(* CODESYS project vertical_levitation_control_new.library
   TcLibraryId: TE140x Module Vendor|vertical_levitation_control_new|0.0.0.21
   Company: TE140x Module Vendor
   Title: vertical_levitation_control_new
   Placeholder: vertical_levitation_control_new
   Version: 0.0.0.21

Project tree, tasks and I/O mapping:
  POUs/
    function block FB_vertical_levitation_control_new [ST]: FB_exit, FB_init, nHResult, eInitExceptionHandling, eUpdateExceptionHandling, nExceptionCnt, stActiveException, bInitialized, bExecute
    TcCOM Wrapper/
      function block FB_vertical_levitation_control_new_TcCOM_InitStruct [ST]: FB_init, FB_afterinit, Reinit, FB_exit, eObjectState, nHResult, ipTcComObject, ipADI, nTaskOid, nTaskPriority, nTaskCycleTimeNs, nTaskPort, nTaskSortOrder, eTraceLevelMax, eModuleCaller, eCallerVerification, eStepSizeAdaptation, eExecutionSequence, bExecute, eAccessLockState, eInitExceptionHandling, eUpdateExceptionHandling, stModuleBuildInfo, bInitialized, nSkippedExecutionCount, stLibraryInfo, stModuleInfo, stModuleGeneratorInfo, stSimulinkModelInfo, evertical_levitation_control_new_P_Sharing, nvertical_levitation_control_new_P_Definer, stvertical_levitation_control_new_P, fSimulationTime, nCycleCount, nExceptionCount, stExceptionInfo
  DUTs/
    data type ST_FB_vertical_levitation_control_new_FB_Main
    data type ST_FB_vertical_levitation_control_new_FB_exit
    data type ST_FB_vertical_levitation_control_new_FB_init
    data type ST_GetSet_HRESULT
    data type E_FpExcptCtrlSetEx
    data type ST_GetSet_E_FpExcptCtrlSetEx
    data type ST_GetSet_ULINT
    data type ST_ExceptionInfo
    data type ST_GetSet_ST_ExceptionInfo
    data type ST_GetSet_BOOL
    data type T_matrix3xdouble
    data type T_matrix2xdouble
    data type T_matrix4xdouble
    data type E_SimTimeStep
    data type E_SolverMode
    data type E_ssMatrixType
    data type ST_RTWRTModelMethodsInfo
    data type E_slJmBdControl
    data type ST_ssSolverInfo
    data type T_matrix8xdouble
    data type T_matrix5xdouble
    data type T_matrix4xlogical
    data type T_matrix8xlogical
    data type ST_B_MATLABFunction_vertical_levitation_control_new_T
    data type ST_B_vertical_levitation_control_new_T
    data type T_ZCSigState
    data type T_matrix4xZCSigState
    data type ST_PrevZCX_vertical_levitation_control_new_T
    data type ST_X_vertical_levitation_control_new_T
    data type ST_ExtU_vertical_levitation_control_new_T
    data type ST_ExtY_vertical_levitation_control_new_T
    data type T_matrix4xbool
    data type ST_XDis_vertical_levitation_control_new_T
    data type T_matrix20xdouble
    data type T_matrix20x4xdouble
    data type PLREAL
    data type T_matrix4xdoublepointer
    data type ST_ODE4_IntgData
    data type ST_DW_vertical_levitation_control_new_T
    data type ST_x08a7a7bbd0e5d629f7d70ceec84eacfe
    data type ST_xf09845edab6c83520d8d57def6d6fe1c
    data type ST_RT_MODEL_vertical_levitation_control_new_T
    data type T_matrix53xdouble
    data type T_matrix1007xdouble
    data type T_matrix19xdouble
    data type T_matrix380xdouble
    data type T_matrix3xlogical
    data type ST_P_vertical_levitation_control_new_T
    data type E_ModuleCaller
    data type E_CallerVerification
    data type E_StepSizeAdaptation
    data type E_ExecutionSequence1
    data type E_FpExcptCtrlSet
    data type ST_TcMatSim_ModuleGeneratorInfo
    data type ST_TcMatSim_SimulinkModelInfo
    data type E_ParameterSharingType
    data type ST_FB_vertical_levitation_control_new_TcCOM_InitStruct
    data type ST_FB_vertical_levitation_control_new_TcCOM_InitStruct_FB_init
    data type ST_FB_vertical_levitation_control_new_TcCOM_InitStruct_FB_afterinit
    data type ST_FB_vertical_levitation_control_new_TcCOM_InitStruct_Reinit
    data type ST_FB_vertical_levitation_control_new_TcCOM_InitStruct_FB_Main
    data type ST_FB_vertical_levitation_control_new_TcCOM_InitStruct_FB_exit
    data type ST_GetSet_TCOM_STATE
    data type ST_GetSet_ITComObject
    data type ST_GetSet_ITcADI
    data type ST_vertical_levitation_control_new_U_T
    data type ST_vertical_levitation_control_new_Y_T
    data type ST_vertical_levitation_control_new_X_T
    data type ST_vertical_levitation_control_new_DW_T
    data type ST_GetSet_OTCID
    data type ST_GetSet_UDINT
    data type ST_GetSet_UINT
    data type ST_GetSet_TcTraceLevel
    data type ST_GetSet_E_ModuleCaller
    data type ST_GetSet_E_CallerVerification
    data type ST_GetSet_E_StepSizeAdaptation
    data type ST_GetSet_E_ExecutionSequence1
    data type ST_GetSet_E_FpExcptCtrlSet
    data type ST_ModuleBuildInfo
    data type ST_GetSet_ST_ModuleBuildInfo
    data type ST_LibraryInfo
    data type ST_GetSet_ST_LibraryInfo
    data type ST_ModuleInfo
    data type ST_GetSet_ST_ModuleInfo
    data type ST_GetSet_ST_TcMatSim_ModuleGeneratorInfo
    data type ST_GetSet_ST_TcMatSim_SimulinkModelInfo
    data type ST_GetSet_E_ParameterSharingType
    data type ST_GetSet_ST_P_vertical_levitation_control_new_T
    data type ST_GetSet_LREAL
  Version/
    global variables Global_Version
*)

// DUTs/ST_FB_vertical_levitation_control_new_FB_Main
{attribute 'TcIecLibraryType'}
{attribute 'hide'}
TYPE ST_FB_vertical_levitation_control_new_FB_Main : 
	STRUCT
		{attribute 'GUID' := '18071995-0000-0000-0000-000000000018'}
		pInst : PVOID;
		result : BOOL;
		 {attribute 'hide'}
		_reserved1 : UINT_24_56;
	END_STRUCT
END_TYPE

// DUTs/ST_FB_vertical_levitation_control_new_FB_exit
{attribute 'TcIecLibraryType'}
{attribute 'hide'}
TYPE ST_FB_vertical_levitation_control_new_FB_exit : 
	STRUCT
		{attribute 'GUID' := '18071995-0000-0000-0000-000000000018'}
		pInst : PVOID;
		bInCopyCode : BOOL;
		result : BOOL;
		 {attribute 'hide'}
		_reserved1 : UINT_16_48;
	END_STRUCT
END_TYPE

// DUTs/ST_FB_vertical_levitation_control_new_FB_init
{attribute 'TcIecLibraryType'}
{attribute 'hide'}
TYPE ST_FB_vertical_levitation_control_new_FB_init : 
	STRUCT
		{attribute 'GUID' := '18071995-0000-0000-0000-000000000018'}
		pInst : PVOID;
		bInitRetains : BOOL;
		bInCopyCode : BOOL;
		result : BOOL;
		 {attribute 'hide'}
		_reserved1 : UINT_8_40;
	END_STRUCT
END_TYPE

// DUTs/ST_GetSet_HRESULT
{attribute 'TcIecLibraryType'}
{attribute 'hide'}
TYPE ST_GetSet_HRESULT : 
	STRUCT
		{attribute 'GUID' := '18071995-0000-0000-0000-000000000018'}
		pInst : PVOID;
		{attribute 'GUID' := '18071995-0000-0000-0000-000000000019'}
		nParam : HRESULT;
		 {attribute 'hide'}
		_reserved1 : UINT_0_32;
	END_STRUCT
END_TYPE

// DUTs/E_FpExcptCtrlSetEx
(* Generated from type 'TcMgSdk.FpExcptCtrlSetEx' *)
{attribute 'TcIecLibraryType'}
TYPE E_FpExcptCtrlSetEx : (
	CallerExceptions:=1, 	(* Use the floating point exception settings provided by the caller *)
	ThrowExceptions:=3, 	(* Enable floating point exceptions on invalid operations and divisions by zero *)
	SuppressExceptions:=13, 	(* Disable floating point exceptions. *)
	LogExceptions:=19, 	(* Log exception information. *)
	LogAndHold:=51, 	(* Log exception information and puase execution of the cyclic code after completion of the actual cycle *)
	LogAndCatch:=83, 	(* Log exception information and immediately terminate execution of the cyclic code. Reinitialization is required to restart. *)
	LogAndDump:=147, 	(* Log exception information, create a dump file with detailed exception information and try to continue execution of the cyclic code *)
	LogHoldAndDump:=179, 	(* Log exception information, create a dump file with detailed exception information and puase execution of the cyclic code after completion of the actual cycle *)
	LogCatchAndDump:=211	(* Log exception information, create a dump file with detailed exception information and immediately terminate execution of the cyclic code. Reinitialization is required to restart. *)
) USINT;
END_TYPE

// DUTs/ST_GetSet_E_FpExcptCtrlSetEx
{attribute 'TcIecLibraryType'}
{attribute 'hide'}
TYPE ST_GetSet_E_FpExcptCtrlSetEx : 
	STRUCT
		{attribute 'GUID' := '18071995-0000-0000-0000-000000000018'}
		pInst : PVOID;
		eParam : E_FpExcptCtrlSetEx;
		 {attribute 'hide'}
		_reserved1 : UINT_24_56;
	END_STRUCT
END_TYPE

// DUTs/ST_GetSet_ULINT
{attribute 'TcIecLibraryType'}
{attribute 'hide'}
TYPE ST_GetSet_ULINT : 
	STRUCT
		{attribute 'GUID' := '18071995-0000-0000-0000-000000000018'}
		pInst : PVOID;
		nParam : ULINT;
	END_STRUCT
END_TYPE

// DUTs/ST_ExceptionInfo
(* Generated from type 'TcMgSdk.ExceptionInfo' *)
{attribute 'TcIecLibraryType'}
TYPE ST_ExceptionInfo : 
	STRUCT
		(* Generated from item 'ExceptionCode' *)
		nExceptionCode : DINT;
		(* Generated from item 'TmxName' *)
		{attribute 'GUID' := '18071995-0000-0000-0000-00010000007F'}
		sTmxName : STRING(127);
		(* Generated from item 'TmxVersion' *)
		nTmxVersion : ARRAY [0..3] OF UDINT;
		(* Generated from item 'InstructionAddr' *)
		nInstructionAddr : UDINT;
		(* Generated from item 'ReturnAddr' *)
		nReturnAddr : ARRAY [0..3] OF UDINT;
		(* Generated from item 'DumpCreated' *)
		bDumpCreated : BOOL;
		 {attribute 'hide'}
		_reserved1 : ARRAY [1..3] OF USINT;
	END_STRUCT
END_TYPE

// DUTs/ST_GetSet_ST_ExceptionInfo
{attribute 'TcIecLibraryType'}
{attribute 'hide'}
TYPE ST_GetSet_ST_ExceptionInfo : 
	STRUCT
		{attribute 'GUID' := '18071995-0000-0000-0000-000000000018'}
		pInst : PVOID;
		stParam : ST_ExceptionInfo;
		 {attribute 'hide'}
		_reserved1 : UINT_0_32;
	END_STRUCT
END_TYPE

// DUTs/ST_GetSet_BOOL
{attribute 'TcIecLibraryType'}
{attribute 'hide'}
TYPE ST_GetSet_BOOL : 
	STRUCT
		{attribute 'GUID' := '18071995-0000-0000-0000-000000000018'}
		pInst : PVOID;
		bParam : BOOL;
		 {attribute 'hide'}
		_reserved1 : UINT_24_56;
	END_STRUCT
END_TYPE

// DUTs/T_matrix3xdouble
(* Generated from type 'matrix3xdouble' *)
{attribute 'TcIecLibraryType'}
TYPE T_matrix3xdouble : ARRAY [0..2] OF LREAL;
END_TYPE

// DUTs/T_matrix2xdouble
(* Generated from type 'matrix2xdouble' *)
{attribute 'TcIecLibraryType'}
TYPE T_matrix2xdouble : ARRAY [0..1] OF LREAL;
END_TYPE

// DUTs/T_matrix4xdouble
(* Generated from type 'matrix4xdouble' *)
{attribute 'TcIecLibraryType'}
TYPE T_matrix4xdouble : ARRAY [0..3] OF LREAL;
END_TYPE

// DUTs/E_SimTimeStep
(* Generated from type 'SimTimeStep' *)
{attribute 'TcIecLibraryType'}
{attribute 'qualified_only' := 'true'}
TYPE E_SimTimeStep : (MINOR_TIME_STEP:=0, MAJOR_TIME_STEP:=1) DINT;
END_TYPE

// DUTs/E_SolverMode
(* Generated from type 'SolverMode' *)
{attribute 'TcIecLibraryType'}
{attribute 'qualified_only' := 'true'}
TYPE E_SolverMode : (SOLVER_MODE_AUTO:=0, SOLVER_MODE_SINGLETASKING:=1, SOLVER_MODE_MULTITASKING:=2) DINT;
END_TYPE

// DUTs/E_ssMatrixType
(* Generated from type 'ssMatrixType' *)
{attribute 'TcIecLibraryType'}
{attribute 'qualified_only' := 'true'}
TYPE E_ssMatrixType : (SS_MATRIX_NONE:=0, SS_MATRIX_CONSTANT:=1, SS_MATRIX_TIMEDEP:=2, SS_MATRIX_STATEDEP:=3) DINT;
END_TYPE

// DUTs/ST_RTWRTModelMethodsInfo
(* Generated from type 'RTWRTModelMethodsInfo' *)
{attribute 'TcIecLibraryType'}
TYPE ST_RTWRTModelMethodsInfo : 
	STRUCT
		(* Generated from item 'rtModelPtr' *)
		{attribute 'GUID' := '18071995-0000-0000-0000-000000000018'}
		prtModelPtr : PVOID;
		(* Generated from item 'rtmInitSizesFcn' *)
		{attribute 'GUID' := '18071995-0000-0000-0000-000000000018'}
		prtmInitSizesFcn : PVOID;
		(* Generated from item 'rtmInitSampTimesFcn' *)
		{attribute 'GUID' := '18071995-0000-0000-0000-000000000018'}
		prtmInitSampTimesFcn : PVOID;
		(* Generated from item 'rtmStartFcn' *)
		{attribute 'GUID' := '18071995-0000-0000-0000-000000000018'}
		prtmStartFcn : PVOID;
		(* Generated from item 'rtmOutputsFcn' *)
		{attribute 'GUID' := '18071995-0000-0000-0000-000000000018'}
		prtmOutputsFcn : PVOID;
		(* Generated from item 'rtmUpdateFcn' *)
		{attribute 'GUID' := '18071995-0000-0000-0000-000000000018'}
		prtmUpdateFcn : PVOID;
		(* Generated from item 'rtmDervisFcn' *)
		{attribute 'GUID' := '18071995-0000-0000-0000-000000000018'}
		prtmDervisFcn : PVOID;
		(* Generated from item 'rtmProjectionFcn' *)
		{attribute 'GUID' := '18071995-0000-0000-0000-000000000018'}
		prtmProjectionFcn : PVOID;
		(* Generated from item 'rtmMassMatrixFcn' *)
		{attribute 'GUID' := '18071995-0000-0000-0000-000000000018'}
		prtmMassMatrixFcn : PVOID;
		(* Generated from item 'rtmForcingFunctionFcn' *)
		{attribute 'GUID' := '18071995-0000-0000-0000-000000000018'}
		prtmForcingFunctionFcn : PVOID;
		(* Generated from item 'rtmTerminateFcn' *)
		{attribute 'GUID' := '18071995-0000-0000-0000-000000000018'}
		prtmTerminateFcn : PVOID;
		(* Generated from item 'rtmDiscreteEventsFcn' *)
		{attribute 'GUID' := '18071995-0000-0000-0000-000000000018'}
		prtmDiscreteEventsFcn : PVOID;
	END_STRUCT
END_TYPE

// DUTs/E_slJmBdControl
(* Generated from type 'slJmBdControl' *)
{attribute 'TcIecLibraryType'}
{attribute 'qualified_only' := 'true'}
TYPE E_slJmBdControl : (SL_JM_BD_AUTO:=0, SL_JM_BD_SPARSE_PERTURBATION:=1, SL_JM_BD_FULL_PERTURBATION:=2, SL_JM_BD_SPARSE_ANALYTICAL:=3, SL_JM_BD_FULL_ANALYTICAL:=4) DINT;
END_TYPE

// DUTs/ST_ssSolverInfo
(* Generated from type 'ssSolverInfo' *)
{attribute 'TcIecLibraryType'}
TYPE ST_ssSolverInfo : 
	STRUCT
		(* Generated from item 'rtModelPtr' *)
		{attribute 'GUID' := '18071995-0000-0000-0000-000000000018'}
		prtModelPtr : PVOID;
		simTimeStepPtr : POINTER TO E_SimTimeStep;
		(* Generated from item 'solverData' *)
		{attribute 'GUID' := '18071995-0000-0000-0000-000000000018'}
		psolverData : PVOID;
		solverName : POINTER TO SINT;
		(* Generated from item 'isVariableStepSolver' *)
		bisVariableStepSolver : BOOL;
		(* Generated from item 'solverNeedsReset' *)
		bsolverNeedsReset : BOOL;
		 {attribute 'hide'}
		_reserved1 : UINT;
		(* Generated from item 'solverMode' *)
		esolverMode : E_SolverMode;
		(* Generated from item 'solverStopTime' *)
		fsolverStopTime : LREAL;
		stepSizePtr : POINTER TO LREAL;
		(* Generated from item 'minStepSize' *)
		fminStepSize : LREAL;
		(* Generated from item 'maxStepSize' *)
		fmaxStepSize : LREAL;
		(* Generated from item 'fixedStepSize' *)
		ffixedStepSize : LREAL;
		(* Generated from item 'solverShapePreserveControl' *)
		nsolverShapePreserveControl : DINT;
		(* Generated from item 'solverMaxConsecutiveMinStep' *)
		nsolverMaxConsecutiveMinStep : DINT;
		(* Generated from item 'maxNumMinSteps' *)
		nmaxNumMinSteps : DINT;
		(* Generated from item 'solverMaxOrder' *)
		nsolverMaxOrder : DINT;
		(* Generated from item 'solverConsecutiveZCsStepRelTol' *)
		fsolverConsecutiveZCsStepRelTol : LREAL;
		(* Generated from item 'solverMaxConsecutiveZCs' *)
		nsolverMaxConsecutiveZCs : DINT;
		(* Generated from item 'solverExtrapolationOrder' *)
		nsolverExtrapolationOrder : DINT;
		(* Generated from item 'solverNumberNewtonIterations' *)
		nsolverNumberNewtonIterations : DINT;
		(* Generated from item 'solverRefineFactor' *)
		nsolverRefineFactor : DINT;
		(* Generated from item 'solverRelTol' *)
		fsolverRelTol : LREAL;
		(* Generated from item 'unused_real_T_1' *)
		funused_real_T_1 : LREAL;
		dXPtr : POINTER TO POINTER TO LREAL;
		tPtr : POINTER TO POINTER TO LREAL;
		numContStatesPtr : POINTER TO DINT;
		contStatesPtr : POINTER TO POINTER TO LREAL;
		numPeriodicContStatesPtr : POINTER TO DINT;
		periodicContStateIndicesPtr : POINTER TO POINTER TO DINT;
		periodicContStateRangesPtr : POINTER TO POINTER TO LREAL;
		zcSignalVector : POINTER TO LREAL;
		zcEventsVector : POINTER TO USINT;
		zcSignalAttrib : POINTER TO USINT;
		(* Generated from item 'zcSignalVectorLength' *)
		nzcSignalVectorLength : DINT;
		 {attribute 'hide'}
		_reserved2 : UINT_0_32;
		reserved : POINTER TO USINT;
		(* Generated from item 'foundContZcEvents' *)
		bfoundContZcEvents : BOOL;
		(* Generated from item 'isAtLeftPostOfContZcEvent' *)
		bisAtLeftPostOfContZcEvent : BOOL;
		(* Generated from item 'isAtRightPostOfContZcEvent' *)
		bisAtRightPostOfContZcEvent : BOOL;
		(* Generated from item 'adaptiveZcDetection' *)
		badaptiveZcDetection : BOOL;
		(* Generated from item 'numZcSignals' *)
		nnumZcSignals : DINT;
		(* Generated from item 'stateProjection' *)
		bstateProjection : BOOL;
		(* Generated from item 'robustResetMethod' *)
		brobustResetMethod : BOOL;
		(* Generated from item 'updateJacobianAtReset' *)
		bupdateJacobianAtReset : BOOL;
		(* Generated from item 'consistencyChecking' *)
		bconsistencyChecking : BOOL;
		(* Generated from item 'massMatrixType' *)
		emassMatrixType : E_ssMatrixType;
		(* Generated from item 'massMatrixNzMax' *)
		nmassMatrixNzMax : DINT;
		 {attribute 'hide'}
		_reserved3 : UINT_0_32;
		massMatrixIr : POINTER TO DINT;
		massMatrixJc : POINTER TO DINT;
		massMatrixPr : POINTER TO LREAL;
		errStatusPtr : POINTER TO POINTER TO SINT;
		modelMethodsPtr : POINTER TO ST_RTWRTModelMethodsInfo;
		(* Generated from item 'zcThreshold' *)
		fzcThreshold : LREAL;
		(* Generated from item 'reserved_1' *)
		nreserved_1 : DINT;
		(* Generated from item 'consecutiveZCsError' *)
		nconsecutiveZCsError : DINT;
		(* Generated from item 'CTOutputIncnstWithState' *)
		bCTOutputIncnstWithState : BOOL;
		(* Generated from item 'isComputingJacobian' *)
		bisComputingJacobian : BOOL;
		 {attribute 'hide'}
		_reserved4 : UINT;
		(* Generated from item 'solverJacobianMethodControl' *)
		esolverJacobianMethodControl : E_slJmBdControl;
		(* Generated from item 'ignoredZcDiagnostic' *)
		nignoredZcDiagnostic : DINT;
		(* Generated from item 'maskedZcDiagnostic' *)
		nmaskedZcDiagnostic : DINT;
		(* Generated from item 'isOutputMethodComputed' *)
		bisOutputMethodComputed : BOOL;
		 {attribute 'hide'}
		_reserved5 : ARRAY [1..3] OF USINT;
		(* Generated from item 'maxZcBracketingIterations' *)
		nmaxZcBracketingIterations : DINT;
		(* Generated from item 'isMinorTimeStepWithModeChange' *)
		bisMinorTimeStepWithModeChange : BOOL;
		 {attribute 'hide'}
		_reserved6 : ARRAY [1..3] OF USINT;
		(* Generated from item 'maxZcPerStep' *)
		nmaxZcPerStep : DINT;
		zcSignalPtr : POINTER TO POINTER TO LREAL;
		(* Generated from item 'contStateDisabledPtr' *)
		bcontStateDisabledPtr : POINTER TO POINTER TO BOOL;
		(* Generated from item 'isContModeFrozen' *)
		bisContModeFrozen : BOOL;
		 {attribute 'hide'}
		_reserved7 : ARRAY [1..7] OF USINT;
	END_STRUCT
END_TYPE

// DUTs/T_matrix8xdouble
(* Generated from type 'matrix8xdouble' *)
{attribute 'TcIecLibraryType'}
TYPE T_matrix8xdouble : ARRAY [0..7] OF LREAL;
END_TYPE

// DUTs/T_matrix5xdouble
(* Generated from type 'matrix5xdouble' *)
{attribute 'TcIecLibraryType'}
TYPE T_matrix5xdouble : ARRAY [0..4] OF LREAL;
END_TYPE

// DUTs/T_matrix4xlogical
(* Generated from type 'matrix4xlogical' *)
{attribute 'TcIecLibraryType'}
{attribute 'BaseTypeGUID' := '18071995-0000-0000-0000-000000000030'}
TYPE T_matrix4xlogical : ARRAY [0..3] OF BOOL;
END_TYPE

// DUTs/T_matrix8xlogical
(* Generated from type 'matrix8xlogical' *)
{attribute 'TcIecLibraryType'}
{attribute 'BaseTypeGUID' := '18071995-0000-0000-0000-000000000030'}
TYPE T_matrix8xlogical : ARRAY [0..7] OF BOOL;
END_TYPE

// DUTs/ST_B_MATLABFunction_vertical_levitation_control_new_T
(* Generated from type 'B_MATLABFunction_vertical_levitation_control_new_T' *)
{attribute 'TcIecLibraryType'}
TYPE ST_B_MATLABFunction_vertical_levitation_control_new_T : 
	STRUCT
		(* Generated from item 'y' *)
		ay : T_matrix8xdouble;
	END_STRUCT
END_TYPE

// DUTs/ST_B_vertical_levitation_control_new_T
(* Generated from type 'B_vertical_levitation_control_new_T' *)
{attribute 'TcIecLibraryType'}
TYPE ST_B_vertical_levitation_control_new_T : 
	STRUCT
		(* Generated from item 'UnitDelay' *)
		aUnitDelay : T_matrix4xdouble;
		(* Generated from item 'Switch1' *)
		aSwitch1 : T_matrix4xdouble;
		(* Generated from item 'Switch1_d' *)
		aSwitch1_d : T_matrix4xdouble;
		(* Generated from item 'Gain3' *)
		fGain3 : LREAL;
		(* Generated from item 'Gain7' *)
		fGain7 : LREAL;
		(* Generated from item 'Switch2' *)
		aSwitch2 : T_matrix4xdouble;
		(* Generated from item 'select_maxs' *)
		aselect_maxs : T_matrix4xdouble;
		(* Generated from item 'Delay' *)
		aDelay : T_matrix3xdouble;
		(* Generated from item 'UnitDelay1' *)
		fUnitDelay1 : LREAL;
		(* Generated from item 'FilterCoefficient' *)
		fFilterCoefficient : LREAL;
		(* Generated from item 'Saturation' *)
		fSaturation : LREAL;
		(* Generated from item 'Gain10' *)
		fGain10 : LREAL;
		(* Generated from item 'Integrator' *)
		fIntegrator : LREAL;
		(* Generated from item 'Filtertotgain' *)
		fFiltertotgain : LREAL;
		(* Generated from item 'Add4' *)
		fAdd4 : LREAL;
		(* Generated from item 'UnitDelay1_h' *)
		fUnitDelay1_h : LREAL;
		(* Generated from item 'Add4_f' *)
		fAdd4_f : LREAL;
		(* Generated from item 'UnitDelay1_i' *)
		fUnitDelay1_i : LREAL;
		(* Generated from item 'Add4_d' *)
		fAdd4_d : LREAL;
		(* Generated from item 'UnitDelay1_ie' *)
		fUnitDelay1_ie : LREAL;
		(* Generated from item 'Add4_m' *)
		fAdd4_m : LREAL;
		(* Generated from item 'UnitDelay1_l' *)
		fUnitDelay1_l : LREAL;
		(* Generated from item 'Add4_c' *)
		fAdd4_c : LREAL;
		(* Generated from item 'UnitDelay1_o' *)
		fUnitDelay1_o : LREAL;
		(* Generated from item 'Add4_a' *)
		fAdd4_a : LREAL;
		(* Generated from item 'UnitDelay1_iy' *)
		fUnitDelay1_iy : LREAL;
		(* Generated from item 'Add4_l' *)
		fAdd4_l : LREAL;
		(* Generated from item 'UnitDelay1_a' *)
		fUnitDelay1_a : LREAL;
		(* Generated from item 'Switch1_d5' *)
		fSwitch1_d5 : LREAL;
		(* Generated from item 'Gain12' *)
		fGain12 : LREAL;
		(* Generated from item 'Integrator_g' *)
		fIntegrator_g : LREAL;
		(* Generated from item 'K_D_roll' *)
		fK_D_roll : LREAL;
		(* Generated from item 'Filterrollgain' *)
		fFilterrollgain : LREAL;
		(* Generated from item 'TSamp' *)
		fTSamp : LREAL;
		(* Generated from item 'Diff' *)
		fDiff : LREAL;
		(* Generated from item 'Add4_me' *)
		fAdd4_me : LREAL;
		(* Generated from item 'UnitDelay1_ht' *)
		fUnitDelay1_ht : LREAL;
		(* Generated from item 'Add4_k' *)
		fAdd4_k : LREAL;
		(* Generated from item 'UnitDelay1_oe' *)
		fUnitDelay1_oe : LREAL;
		(* Generated from item 'Add4_ab' *)
		fAdd4_ab : LREAL;
		(* Generated from item 'UnitDelay1_d' *)
		fUnitDelay1_d : LREAL;
		(* Generated from item 'Add4_b' *)
		fAdd4_b : LREAL;
		(* Generated from item 'UnitDelay1_n' *)
		fUnitDelay1_n : LREAL;
		(* Generated from item 'Add4_i' *)
		fAdd4_i : LREAL;
		(* Generated from item 'UnitDelay1_f' *)
		fUnitDelay1_f : LREAL;
		(* Generated from item 'Add4_h' *)
		fAdd4_h : LREAL;
		(* Generated from item 'UnitDelay1_g' *)
		fUnitDelay1_g : LREAL;
		(* Generated from item 'Add4_be' *)
		fAdd4_be : LREAL;
		(* Generated from item 'UnitDelay1_k' *)
		fUnitDelay1_k : LREAL;
		(* Generated from item 'Switch1_m' *)
		fSwitch1_m : LREAL;
		(* Generated from item 'Gain13' *)
		fGain13 : LREAL;
		(* Generated from item 'Integrator_i' *)
		fIntegrator_i : LREAL;
		(* Generated from item 'Filterpitgain' *)
		fFilterpitgain : LREAL;
		(* Generated from item 'Add4_n' *)
		fAdd4_n : LREAL;
		(* Generated from item 'UnitDelay1_fu' *)
		fUnitDelay1_fu : LREAL;
		(* Generated from item 'Add4_g' *)
		fAdd4_g : LREAL;
		(* Generated from item 'UnitDelay1_ha' *)
		fUnitDelay1_ha : LREAL;
		(* Generated from item 'Add4_dq' *)
		fAdd4_dq : LREAL;
		(* Generated from item 'UnitDelay1_ip' *)
		fUnitDelay1_ip : LREAL;
		(* Generated from item 'Add4_dp' *)
		fAdd4_dp : LREAL;
		(* Generated from item 'UnitDelay1_an' *)
		fUnitDelay1_an : LREAL;
		(* Generated from item 'Add4_p' *)
		fAdd4_p : LREAL;
		(* Generated from item 'UnitDelay1_p' *)
		fUnitDelay1_p : LREAL;
		(* Generated from item 'Add4_kw' *)
		fAdd4_kw : LREAL;
		(* Generated from item 'UnitDelay1_dw' *)
		fUnitDelay1_dw : LREAL;
		(* Generated from item 'Add4_hd' *)
		fAdd4_hd : LREAL;
		(* Generated from item 'UnitDelay1_g1' *)
		fUnitDelay1_g1 : LREAL;
		(* Generated from item 'Switch1_n' *)
		fSwitch1_n : LREAL;
		(* Generated from item 'select_mins' *)
		aselect_mins : T_matrix4xdouble;
		(* Generated from item 'Switch' *)
		fSwitch : LREAL;
		(* Generated from item 'UnitDelay1_m' *)
		fUnitDelay1_m : LREAL;
		(* Generated from item 'FilterCoefficient_l' *)
		fFilterCoefficient_l : LREAL;
		(* Generated from item 'Saturation_p' *)
		fSaturation_p : LREAL;
		(* Generated from item 'Switch1_a' *)
		fSwitch1_a : LREAL;
		(* Generated from item 'UnitDelay1_nr' *)
		fUnitDelay1_nr : LREAL;
		(* Generated from item 'FilterCoefficient_o' *)
		fFilterCoefficient_o : LREAL;
		(* Generated from item 'Saturation_pi' *)
		fSaturation_pi : LREAL;
		(* Generated from item 'Switch2_j' *)
		fSwitch2_j : LREAL;
		(* Generated from item 'F_hemsfinal' *)
		aF_hemsfinal : T_matrix4xdouble;
		(* Generated from item 'Switch2_f' *)
		aSwitch2_f : T_matrix8xdouble;
		(* Generated from item 'Switch_o' *)
		fSwitch_o : LREAL;
		(* Generated from item 'Switch_j' *)
		fSwitch_j : LREAL;
		(* Generated from item 'Switch_k' *)
		fSwitch_k : LREAL;
		(* Generated from item 'Add5' *)
		fAdd5 : LREAL;
		(* Generated from item 'Add6' *)
		fAdd6 : LREAL;
		(* Generated from item 'Gain' *)
		fGain : LREAL;
		(* Generated from item 'UnitDelay2' *)
		fUnitDelay2 : LREAL;
		(* Generated from item 'Sum4' *)
		fSum4 : LREAL;
		(* Generated from item 'Sum5' *)
		fSum5 : LREAL;
		(* Generated from item 'Add5_h' *)
		fAdd5_h : LREAL;
		(* Generated from item 'Add6_g' *)
		fAdd6_g : LREAL;
		(* Generated from item 'Gain_l' *)
		fGain_l : LREAL;
		(* Generated from item 'UnitDelay2_k' *)
		fUnitDelay2_k : LREAL;
		(* Generated from item 'Sum4_p' *)
		fSum4_p : LREAL;
		(* Generated from item 'Sum5_p' *)
		fSum5_p : LREAL;
		(* Generated from item 'Add5_m' *)
		fAdd5_m : LREAL;
		(* Generated from item 'Add6_i' *)
		fAdd6_i : LREAL;
		(* Generated from item 'Gain_l5' *)
		fGain_l5 : LREAL;
		(* Generated from item 'UnitDelay2_d' *)
		fUnitDelay2_d : LREAL;
		(* Generated from item 'Sum4_i' *)
		fSum4_i : LREAL;
		(* Generated from item 'Sum5_b' *)
		fSum5_b : LREAL;
		(* Generated from item 'Add5_o' *)
		fAdd5_o : LREAL;
		(* Generated from item 'Add6_m' *)
		fAdd6_m : LREAL;
		(* Generated from item 'Gain_n' *)
		fGain_n : LREAL;
		(* Generated from item 'UnitDelay2_n' *)
		fUnitDelay2_n : LREAL;
		(* Generated from item 'Sum4_f' *)
		fSum4_f : LREAL;
		(* Generated from item 'Sum5_e' *)
		fSum5_e : LREAL;
		(* Generated from item 'Add5_f' *)
		fAdd5_f : LREAL;
		(* Generated from item 'Add6_my' *)
		fAdd6_my : LREAL;
		(* Generated from item 'Gain_ne' *)
		fGain_ne : LREAL;
		(* Generated from item 'UnitDelay2_h' *)
		fUnitDelay2_h : LREAL;
		(* Generated from item 'Sum4_a' *)
		fSum4_a : LREAL;
		(* Generated from item 'Sum5_n' *)
		fSum5_n : LREAL;
		(* Generated from item 'Add5_j' *)
		fAdd5_j : LREAL;
		(* Generated from item 'Add6_l' *)
		fAdd6_l : LREAL;
		(* Generated from item 'Gain_a' *)
		fGain_a : LREAL;
		(* Generated from item 'UnitDelay2_di' *)
		fUnitDelay2_di : LREAL;
		(* Generated from item 'Sum4_pc' *)
		fSum4_pc : LREAL;
		(* Generated from item 'Sum5_g' *)
		fSum5_g : LREAL;
		(* Generated from item 'Add5_k' *)
		fAdd5_k : LREAL;
		(* Generated from item 'Add6_f' *)
		fAdd6_f : LREAL;
		(* Generated from item 'Gain_f' *)
		fGain_f : LREAL;
		(* Generated from item 'UnitDelay2_dw' *)
		fUnitDelay2_dw : LREAL;
		(* Generated from item 'Sum4_d' *)
		fSum4_d : LREAL;
		(* Generated from item 'Sum5_k' *)
		fSum5_k : LREAL;
		(* Generated from item 'Add5_ma' *)
		fAdd5_ma : LREAL;
		(* Generated from item 'Add6_n' *)
		fAdd6_n : LREAL;
		(* Generated from item 'Gain_d' *)
		fGain_d : LREAL;
		(* Generated from item 'UnitDelay2_l' *)
		fUnitDelay2_l : LREAL;
		(* Generated from item 'Sum4_d1' *)
		fSum4_d1 : LREAL;
		(* Generated from item 'Sum5_f' *)
		fSum5_f : LREAL;
		(* Generated from item 'Add5_c' *)
		fAdd5_c : LREAL;
		(* Generated from item 'Add6_mq' *)
		fAdd6_mq : LREAL;
		(* Generated from item 'Gain_k' *)
		fGain_k : LREAL;
		(* Generated from item 'UnitDelay2_o' *)
		fUnitDelay2_o : LREAL;
		(* Generated from item 'Sum4_io' *)
		fSum4_io : LREAL;
		(* Generated from item 'Sum5_j' *)
		fSum5_j : LREAL;
		(* Generated from item 'Add5_op' *)
		fAdd5_op : LREAL;
		(* Generated from item 'Add6_o' *)
		fAdd6_o : LREAL;
		(* Generated from item 'Gain_p' *)
		fGain_p : LREAL;
		(* Generated from item 'UnitDelay2_f' *)
		fUnitDelay2_f : LREAL;
		(* Generated from item 'Sum4_di' *)
		fSum4_di : LREAL;
		(* Generated from item 'Sum5_p3' *)
		fSum5_p3 : LREAL;
		(* Generated from item 'Add5_e' *)
		fAdd5_e : LREAL;
		(* Generated from item 'Add6_k' *)
		fAdd6_k : LREAL;
		(* Generated from item 'Gain_m' *)
		fGain_m : LREAL;
		(* Generated from item 'UnitDelay2_c' *)
		fUnitDelay2_c : LREAL;
		(* Generated from item 'Sum4_e' *)
		fSum4_e : LREAL;
		(* Generated from item 'Sum5_jo' *)
		fSum5_jo : LREAL;
		(* Generated from item 'Add5_kt' *)
		fAdd5_kt : LREAL;
		(* Generated from item 'Add6_d' *)
		fAdd6_d : LREAL;
		(* Generated from item 'Gain_p5' *)
		fGain_p5 : LREAL;
		(* Generated from item 'UnitDelay2_b' *)
		fUnitDelay2_b : LREAL;
		(* Generated from item 'Sum4_c' *)
		fSum4_c : LREAL;
		(* Generated from item 'Sum5_c' *)
		fSum5_c : LREAL;
		(* Generated from item 'Add5_g' *)
		fAdd5_g : LREAL;
		(* Generated from item 'Add6_dl' *)
		fAdd6_dl : LREAL;
		(* Generated from item 'Gain_n2' *)
		fGain_n2 : LREAL;
		(* Generated from item 'UnitDelay2_g' *)
		fUnitDelay2_g : LREAL;
		(* Generated from item 'Sum4_dt' *)
		fSum4_dt : LREAL;
		(* Generated from item 'Sum5_cj' *)
		fSum5_cj : LREAL;
		(* Generated from item 'Add5_gc' *)
		fAdd5_gc : LREAL;
		(* Generated from item 'Add6_a' *)
		fAdd6_a : LREAL;
		(* Generated from item 'Gain_li' *)
		fGain_li : LREAL;
		(* Generated from item 'UnitDelay2_i' *)
		fUnitDelay2_i : LREAL;
		(* Generated from item 'Sum4_k' *)
		fSum4_k : LREAL;
		(* Generated from item 'Sum5_p4' *)
		fSum5_p4 : LREAL;
		(* Generated from item 'Add5_es' *)
		fAdd5_es : LREAL;
		(* Generated from item 'Add6_k2' *)
		fAdd6_k2 : LREAL;
		(* Generated from item 'Gain_i' *)
		fGain_i : LREAL;
		(* Generated from item 'UnitDelay2_n5' *)
		fUnitDelay2_n5 : LREAL;
		(* Generated from item 'Sum4_o' *)
		fSum4_o : LREAL;
		(* Generated from item 'Sum5_po' *)
		fSum5_po : LREAL;
		(* Generated from item 'Add5_l' *)
		fAdd5_l : LREAL;
		(* Generated from item 'Add6_c' *)
		fAdd6_c : LREAL;
		(* Generated from item 'Gain_mr' *)
		fGain_mr : LREAL;
		(* Generated from item 'UnitDelay2_e' *)
		fUnitDelay2_e : LREAL;
		(* Generated from item 'Sum4_p3' *)
		fSum4_p3 : LREAL;
		(* Generated from item 'Sum5_nz' *)
		fSum5_nz : LREAL;
		(* Generated from item 'Add5_je' *)
		fAdd5_je : LREAL;
		(* Generated from item 'Add6_a2' *)
		fAdd6_a2 : LREAL;
		(* Generated from item 'Gain_fh' *)
		fGain_fh : LREAL;
		(* Generated from item 'UnitDelay2_cg' *)
		fUnitDelay2_cg : LREAL;
		(* Generated from item 'Sum4_o5' *)
		fSum4_o5 : LREAL;
		(* Generated from item 'Sum5_d' *)
		fSum5_d : LREAL;
		(* Generated from item 'Add5_b' *)
		fAdd5_b : LREAL;
		(* Generated from item 'Add6_e' *)
		fAdd6_e : LREAL;
		(* Generated from item 'Gain_j' *)
		fGain_j : LREAL;
		(* Generated from item 'UnitDelay2_c5' *)
		fUnitDelay2_c5 : LREAL;
		(* Generated from item 'Sum4_fb' *)
		fSum4_fb : LREAL;
		(* Generated from item 'Sum5_js' *)
		fSum5_js : LREAL;
		(* Generated from item 'Add5_b0' *)
		fAdd5_b0 : LREAL;
		(* Generated from item 'Add6_nn' *)
		fAdd6_nn : LREAL;
		(* Generated from item 'Gain_pn' *)
		fGain_pn : LREAL;
		(* Generated from item 'UnitDelay2_k0' *)
		fUnitDelay2_k0 : LREAL;
		(* Generated from item 'Sum4_pd' *)
		fSum4_pd : LREAL;
		(* Generated from item 'Sum5_m' *)
		fSum5_m : LREAL;
		(* Generated from item 'Add5_fq' *)
		fAdd5_fq : LREAL;
		(* Generated from item 'Add6_i1' *)
		fAdd6_i1 : LREAL;
		(* Generated from item 'Gain_p0' *)
		fGain_p0 : LREAL;
		(* Generated from item 'UnitDelay2_o4' *)
		fUnitDelay2_o4 : LREAL;
		(* Generated from item 'Sum4_kn' *)
		fSum4_kn : LREAL;
		(* Generated from item 'Sum5_a' *)
		fSum5_a : LREAL;
		(* Generated from item 'Add5_mq' *)
		fAdd5_mq : LREAL;
		(* Generated from item 'Add6_j' *)
		fAdd6_j : LREAL;
		(* Generated from item 'Gain_ay' *)
		fGain_ay : LREAL;
		(* Generated from item 'UnitDelay2_hz' *)
		fUnitDelay2_hz : LREAL;
		(* Generated from item 'Sum4_ku' *)
		fSum4_ku : LREAL;
		(* Generated from item 'Sum5_kh' *)
		fSum5_kh : LREAL;
		(* Generated from item 'IsPeak1' *)
		aIsPeak1 : T_matrix4xdouble;
		(* Generated from item 'Switch2_d' *)
		aSwitch2_d : T_matrix4xdouble;
		(* Generated from item 'F_netpostfm' *)
		aF_netpostfm : T_matrix3xdouble;
		(* Generated from item 'Sum' *)
		fSum : LREAL;
		(* Generated from item 'Sum1' *)
		fSum1 : LREAL;
		(* Generated from item 'clamppit' *)
		fclamppit : LREAL;
		(* Generated from item 'Sum_f' *)
		fSum_f : LREAL;
		(* Generated from item 'Sum1_a' *)
		fSum1_a : LREAL;
		(* Generated from item 'clamproll' *)
		fclamproll : LREAL;
		(* Generated from item 'clamptot' *)
		fclamptot : LREAL;
		(* Generated from item 'K_I_tot' *)
		fK_I_tot : LREAL;
		(* Generated from item 'K_I_roll' *)
		fK_I_roll : LREAL;
		(* Generated from item 'K_I_pit' *)
		fK_I_pit : LREAL;
		(* Generated from item 'current_reqf' *)
		fcurrent_reqf : LREAL;
		(* Generated from item 'current_reqb' *)
		fcurrent_reqb : LREAL;
		(* Generated from item 'current_reqf_p' *)
		fcurrent_reqf_p : LREAL;
		(* Generated from item 'current_reqb_o' *)
		fcurrent_reqb_o : LREAL;
		(* Generated from item 'current_reqf_c' *)
		fcurrent_reqf_c : LREAL;
		(* Generated from item 'current_reqb_c' *)
		fcurrent_reqb_c : LREAL;
		(* Generated from item 'current_reqf_h' *)
		fcurrent_reqf_h : LREAL;
		(* Generated from item 'current_reqb_e' *)
		fcurrent_reqb_e : LREAL;
		(* Generated from item 'F_hems' *)
		aF_hems : T_matrix4xdouble;
		(* Generated from item 'Switch2_l' *)
		aSwitch2_l : T_matrix4xdouble;
		(* Generated from item 'Sum5_fo' *)
		fSum5_fo : LREAL;
		(* Generated from item 'Is' *)
		aIs : T_matrix4xdouble;
		(* Generated from item 'satn' *)
		asatn : T_matrix8xdouble;
		(* Generated from item 'airgaps_avg' *)
		aairgaps_avg : T_matrix4xdouble;
		(* Generated from item 'airgap_diff' *)
		fairgap_diff : LREAL;
		(* Generated from item 'tau_x' *)
		ftau_x : LREAL;
		(* Generated from item 'corrected_out' *)
		fcorrected_out : LREAL;
		(* Generated from item 'corrected_out_j' *)
		fcorrected_out_j : LREAL;
		(* Generated from item 'corrected_out_o' *)
		fcorrected_out_o : LREAL;
		(* Generated from item 'F_hems_b' *)
		aF_hems_b : T_matrix4xdouble;
		(* Generated from item 'clamp_tot' *)
		aclamp_tot : T_matrix2xdouble;
		(* Generated from item 'clamp_roll' *)
		aclamp_roll : T_matrix2xdouble;
		(* Generated from item 'clamp_pit' *)
		aclamp_pit : T_matrix2xdouble;
		(* Generated from item 'counter' *)
		acounter : T_matrix5xdouble;
		(* Generated from item 'F_dof_sat' *)
		aF_dof_sat : T_matrix3xdouble;
		(* Generated from item 'sat_fail' *)
		fsat_fail : LREAL;
		(* Generated from item 'q' *)
		fq : LREAL;
		(* Generated from item 'q_c' *)
		fq_c : LREAL;
		(* Generated from item 'q_k' *)
		fq_k : LREAL;
		(* Generated from item 'q_i' *)
		fq_i : LREAL;
		(* Generated from item 'q_g' *)
		fq_g : LREAL;
		(* Generated from item 'q_ke' *)
		fq_ke : LREAL;
		(* Generated from item 'q_b' *)
		fq_b : LREAL;
		(* Generated from item 'q_km' *)
		fq_km : LREAL;
		(* Generated from item 'q_o' *)
		fq_o : LREAL;
		(* Generated from item 'q_a' *)
		fq_a : LREAL;
		(* Generated from item 'q_ag' *)
		fq_ag : LREAL;
		(* Generated from item 'q_d' *)
		fq_d : LREAL;
		(* Generated from item 'q_f' *)
		fq_f : LREAL;
		(* Generated from item 'q_m' *)
		fq_m : LREAL;
		(* Generated from item 'q_n' *)
		fq_n : LREAL;
		(* Generated from item 'q_iy' *)
		fq_iy : LREAL;
		(* Generated from item 'q_h' *)
		fq_h : LREAL;
		(* Generated from item 'q_kmf' *)
		fq_kmf : LREAL;
		(* Generated from item 'q_a3' *)
		fq_a3 : LREAL;
		(* Generated from item 'q_ac' *)
		fq_ac : LREAL;
		(* Generated from item 'q_p' *)
		fq_p : LREAL;
		(* Generated from item 'UnaryMinus' *)
		fUnaryMinus : LREAL;
		(* Generated from item 'UnaryMinus_l' *)
		fUnaryMinus_l : LREAL;
		(* Generated from item 'UnaryMinus_k' *)
		fUnaryMinus_k : LREAL;
		(* Generated from item 'UnaryMinus_b' *)
		fUnaryMinus_b : LREAL;
		(* Generated from item 'UnaryMinus_d' *)
		fUnaryMinus_d : LREAL;
		(* Generated from item 'UnaryMinus_f' *)
		fUnaryMinus_f : LREAL;
		(* Generated from item 'UnaryMinus_k2' *)
		fUnaryMinus_k2 : LREAL;
		(* Generated from item 'UnaryMinus_dc' *)
		fUnaryMinus_dc : LREAL;
		(* Generated from item 'UnaryMinus_m' *)
		fUnaryMinus_m : LREAL;
		(* Generated from item 'UnaryMinus_p' *)
		fUnaryMinus_p : LREAL;
		(* Generated from item 'UnaryMinus_me' *)
		fUnaryMinus_me : LREAL;
		(* Generated from item 'UnaryMinus_l0' *)
		fUnaryMinus_l0 : LREAL;
		(* Generated from item 'UnaryMinus_mg' *)
		fUnaryMinus_mg : LREAL;
		(* Generated from item 'UnaryMinus_o' *)
		fUnaryMinus_o : LREAL;
		(* Generated from item 'UnaryMinus_fu' *)
		fUnaryMinus_fu : LREAL;
		(* Generated from item 'UnaryMinus_e' *)
		fUnaryMinus_e : LREAL;
		(* Generated from item 'UnaryMinus_n' *)
		fUnaryMinus_n : LREAL;
		(* Generated from item 'UnaryMinus_on' *)
		fUnaryMinus_on : LREAL;
		(* Generated from item 'UnaryMinus_a' *)
		fUnaryMinus_a : LREAL;
		(* Generated from item 'UnaryMinus_lr' *)
		fUnaryMinus_lr : LREAL;
		(* Generated from item 'UnaryMinus_mk' *)
		fUnaryMinus_mk : LREAL;
		(* Generated from item 'Integrator2' *)
		aIntegrator2 : T_matrix4xdouble;
		(* Generated from item 'Switch_ka' *)
		aSwitch_ka : T_matrix4xdouble;
		(* Generated from item 'K_P_tot' *)
		fK_P_tot : LREAL;
		(* Generated from item 'Product1' *)
		fProduct1 : LREAL;
		(* Generated from item 'Product1_p' *)
		fProduct1_p : LREAL;
		(* Generated from item 'Product1_i' *)
		fProduct1_i : LREAL;
		(* Generated from item 'TmpSignalConversionAtSFunctionInport1' *)
		aTmpSignalConversionAtSFunctionInport1 : T_matrix3xdouble;
		(* Generated from item 't' *)
		ft : LREAL;
		(* Generated from item 's' *)
		fs : LREAL;
		(* Generated from item 'v' *)
		fv : LREAL;
		(* Generated from item 't_f' *)
		ft_f : LREAL;
		(* Generated from item 's_c' *)
		fs_c : LREAL;
		(* Generated from item 'v_o' *)
		fv_o : LREAL;
		(* Generated from item 'Product4' *)
		fProduct4 : LREAL;
		(* Generated from item 't_h' *)
		ft_h : LREAL;
		(* Generated from item 's_cf' *)
		fs_cf : LREAL;
		(* Generated from item 'v_e' *)
		fv_e : LREAL;
		(* Generated from item 'Product4_c' *)
		fProduct4_c : LREAL;
		(* Generated from item 't_g' *)
		ft_g : LREAL;
		(* Generated from item 's_e' *)
		fs_e : LREAL;
		(* Generated from item 'v_b' *)
		fv_b : LREAL;
		(* Generated from item 'Product4_n' *)
		fProduct4_n : LREAL;
		(* Generated from item 't_i' *)
		ft_i : LREAL;
		(* Generated from item 's_h' *)
		fs_h : LREAL;
		(* Generated from item 'v_j' *)
		fv_j : LREAL;
		(* Generated from item 'Product4_h' *)
		fProduct4_h : LREAL;
		(* Generated from item 't_p' *)
		ft_p : LREAL;
		(* Generated from item 's_f' *)
		fs_f : LREAL;
		(* Generated from item 'v_k' *)
		fv_k : LREAL;
		(* Generated from item 'Product4_d' *)
		fProduct4_d : LREAL;
		(* Generated from item 't_c' *)
		ft_c : LREAL;
		(* Generated from item 's_a' *)
		fs_a : LREAL;
		(* Generated from item 'v_f' *)
		fv_f : LREAL;
		(* Generated from item 't_a' *)
		ft_a : LREAL;
		(* Generated from item 's_o' *)
		fs_o : LREAL;
		(* Generated from item 'v_fk' *)
		fv_fk : LREAL;
		(* Generated from item 't_l' *)
		ft_l : LREAL;
		(* Generated from item 's_b' *)
		fs_b : LREAL;
		(* Generated from item 'v_ex' *)
		fv_ex : LREAL;
		(* Generated from item 'Product4_e' *)
		fProduct4_e : LREAL;
		(* Generated from item 't_lu' *)
		ft_lu : LREAL;
		(* Generated from item 's_fn' *)
		fs_fn : LREAL;
		(* Generated from item 'v_jg' *)
		fv_jg : LREAL;
		(* Generated from item 'Product4_b' *)
		fProduct4_b : LREAL;
		(* Generated from item 't_ch' *)
		ft_ch : LREAL;
		(* Generated from item 's_d' *)
		fs_d : LREAL;
		(* Generated from item 'v_o1' *)
		fv_o1 : LREAL;
		(* Generated from item 'Product4_cg' *)
		fProduct4_cg : LREAL;
		(* Generated from item 't_o' *)
		ft_o : LREAL;
		(* Generated from item 's_hy' *)
		fs_hy : LREAL;
		(* Generated from item 'v_m' *)
		fv_m : LREAL;
		(* Generated from item 'Product4_k' *)
		fProduct4_k : LREAL;
		(* Generated from item 't_j' *)
		ft_j : LREAL;
		(* Generated from item 's_l' *)
		fs_l : LREAL;
		(* Generated from item 'v_mm' *)
		fv_mm : LREAL;
		(* Generated from item 'Product4_n1' *)
		fProduct4_n1 : LREAL;
		(* Generated from item 't_d' *)
		ft_d : LREAL;
		(* Generated from item 's_k' *)
		fs_k : LREAL;
		(* Generated from item 'v_ml' *)
		fv_ml : LREAL;
		(* Generated from item 't_b' *)
		ft_b : LREAL;
		(* Generated from item 's_fd' *)
		fs_fd : LREAL;
		(* Generated from item 'v_d' *)
		fv_d : LREAL;
		(* Generated from item 't_om' *)
		ft_om : LREAL;
		(* Generated from item 's_e3' *)
		fs_e3 : LREAL;
		(* Generated from item 'v_kw' *)
		fv_kw : LREAL;
		(* Generated from item 'Product4_k2' *)
		fProduct4_k2 : LREAL;
		(* Generated from item 't_e' *)
		ft_e : LREAL;
		(* Generated from item 's_p' *)
		fs_p : LREAL;
		(* Generated from item 'v_kl' *)
		fv_kl : LREAL;
		(* Generated from item 'Product4_eq' *)
		fProduct4_eq : LREAL;
		(* Generated from item 't_n' *)
		ft_n : LREAL;
		(* Generated from item 's_g' *)
		fs_g : LREAL;
		(* Generated from item 'v_p' *)
		fv_p : LREAL;
		(* Generated from item 'Product4_ko' *)
		fProduct4_ko : LREAL;
		(* Generated from item 't_dc' *)
		ft_dc : LREAL;
		(* Generated from item 's_g3' *)
		fs_g3 : LREAL;
		(* Generated from item 'Product4_kn' *)
		fProduct4_kn : LREAL;
		(* Generated from item 't_oc' *)
		ft_oc : LREAL;
		(* Generated from item 's_am' *)
		fs_am : LREAL;
		(* Generated from item 'Product4_m' *)
		fProduct4_m : LREAL;
		(* Generated from item 't_bl' *)
		ft_bl : LREAL;
		(* Generated from item 's_kp' *)
		fs_kp : LREAL;
		(* Generated from item 'Integrator_f' *)
		fIntegrator_f : LREAL;
		(* Generated from item 'Product4_b0' *)
		fProduct4_b0 : LREAL;
		(* Generated from item 'u' *)
		fu : LREAL;
		(* Generated from item 'u_b' *)
		fu_b : LREAL;
		(* Generated from item 'u_k' *)
		fu_k : LREAL;
		(* Generated from item 'u_j' *)
		fu_j : LREAL;
		(* Generated from item 'u_d' *)
		fu_d : LREAL;
		(* Generated from item 'u_h' *)
		fu_h : LREAL;
		(* Generated from item 'u_i' *)
		fu_i : LREAL;
		(* Generated from item 'u_p' *)
		fu_p : LREAL;
		(* Generated from item 'u_ba' *)
		fu_ba : LREAL;
		(* Generated from item 'u_id' *)
		fu_id : LREAL;
		(* Generated from item 'u_e' *)
		fu_e : LREAL;
		(* Generated from item 'u_j0' *)
		fu_j0 : LREAL;
		(* Generated from item 'u_i0' *)
		fu_i0 : LREAL;
		(* Generated from item 'u_bj' *)
		fu_bj : LREAL;
		(* Generated from item 'u_iv' *)
		fu_iv : LREAL;
		(* Generated from item 'u_h4' *)
		fu_h4 : LREAL;
		(* Generated from item 'u_kq' *)
		fu_kq : LREAL;
		(* Generated from item 'u_c' *)
		fu_c : LREAL;
		(* Generated from item 'u_a' *)
		fu_a : LREAL;
		(* Generated from item 'u_f' *)
		fu_f : LREAL;
		(* Generated from item 'Final_ON' *)
		aFinal_ON : T_matrix8xdouble;
		(* Generated from item 'Abs1' *)
		aAbs1 : T_matrix4xdouble;
		(* Generated from item 'IntegralGain' *)
		fIntegralGain : LREAL;
		(* Generated from item 'Product3' *)
		fProduct3 : LREAL;
		(* Generated from item 'Product3_l' *)
		fProduct3_l : LREAL;
		(* Generated from item 'Product3_j' *)
		fProduct3_j : LREAL;
		(* Generated from item 'Product3_a' *)
		fProduct3_a : LREAL;
		(* Generated from item 'Product3_b' *)
		fProduct3_b : LREAL;
		(* Generated from item 'Product3_i' *)
		fProduct3_i : LREAL;
		(* Generated from item 'u_dq' *)
		fu_dq : LREAL;
		(* Generated from item 'Product3_c' *)
		fProduct3_c : LREAL;
		(* Generated from item 'Product3_d' *)
		fProduct3_d : LREAL;
		(* Generated from item 'Product3_c5' *)
		fProduct3_c5 : LREAL;
		(* Generated from item 'Product3_d5' *)
		fProduct3_d5 : LREAL;
		(* Generated from item 'Product3_o' *)
		fProduct3_o : LREAL;
		(* Generated from item 'Product3_lu' *)
		fProduct3_lu : LREAL;
		(* Generated from item 'Product4_a' *)
		fProduct4_a : LREAL;
		(* Generated from item 'Product3_f' *)
		fProduct3_f : LREAL;
		(* Generated from item 'Product3_cw' *)
		fProduct3_cw : LREAL;
		(* Generated from item 'Product3_cm' *)
		fProduct3_cm : LREAL;
		(* Generated from item 'Product4_ke' *)
		fProduct4_ke : LREAL;
		(* Generated from item 'Product3_k' *)
		fProduct3_k : LREAL;
		(* Generated from item 'Product4_a4' *)
		fProduct4_a4 : LREAL;
		(* Generated from item 'Product3_h' *)
		fProduct3_h : LREAL;
		(* Generated from item 'Product3_p' *)
		fProduct3_p : LREAL;
		(* Generated from item 'IntegralGain_h' *)
		fIntegralGain_h : LREAL;
		(* Generated from item 'Product3_ph' *)
		fProduct3_ph : LREAL;
		(* Generated from item 'IntegralGain_e' *)
		fIntegralGain_e : LREAL;
		(* Generated from item 'Sign' *)
		fSign : LREAL;
		(* Generated from item 'SignPreSat' *)
		fSignPreSat : LREAL;
		(* Generated from item 'Product4_i' *)
		fProduct4_i : LREAL;
		(* Generated from item 'Product4_ks' *)
		fProduct4_ks : LREAL;
		(* Generated from item 'SignPreSat_g' *)
		fSignPreSat_g : LREAL;
		(* Generated from item 'Product3_je' *)
		fProduct3_je : LREAL;
		(* Generated from item 'Product4_o' *)
		fProduct4_o : LREAL;
		(* Generated from item 'Product4_cr' *)
		fProduct4_cr : LREAL;
		(* Generated from item 'Product3_bw' *)
		fProduct3_bw : LREAL;
		(* Generated from item 'SignPreSat_b' *)
		fSignPreSat_b : LREAL;
		(* Generated from item 'Sign1' *)
		fSign1 : LREAL;
		(* Generated from item 'Product4_ba' *)
		fProduct4_ba : LREAL;
		(* Generated from item 'Delay1' *)
		fDelay1 : REAL;
		(* Generated from item 'fmsatfailordisabled' *)
		ffmsatfailordisabled : REAL;
		(* Generated from item 'hard_disable_fmm' *)
		fhard_disable_fmm : REAL;
		(* Generated from item 'enabled' *)
		nenabled : USINT;
		(* Generated from item 'DataTypeConv2' *)
		nDataTypeConv2 : SINT;
		(* Generated from item 'DataTypeConv1' *)
		nDataTypeConv1 : SINT;
		(* Generated from item 'didfmcausesattofail' *)
		adidfmcausesattofail : T_matrix4xlogical;
		(* Generated from item 'AND3' *)
		bAND3 : BOOL;
		(* Generated from item 'Memory' *)
		bMemory : BOOL;
		(* Generated from item 'AND3_d' *)
		bAND3_d : BOOL;
		(* Generated from item 'Memory_p' *)
		bMemory_p : BOOL;
		(* Generated from item 'AND3_l' *)
		bAND3_l : BOOL;
		(* Generated from item 'Memory_f' *)
		bMemory_f : BOOL;
		(* Generated from item 'y' *)
		_by : BOOL;
		(* Generated from item 'LowerRelop1' *)
		aLowerRelop1 : T_matrix4xlogical;
		(* Generated from item 'UpperRelop' *)
		aUpperRelop : T_matrix4xlogical;
		(* Generated from item 'LowerRelop1_c' *)
		aLowerRelop1_c : T_matrix8xlogical;
		(* Generated from item 'UpperRelop_o' *)
		aUpperRelop_o : T_matrix8xlogical;
		(* Generated from item 'LowerRelop1_e' *)
		aLowerRelop1_e : T_matrix4xlogical;
		(* Generated from item 'AND' *)
		bAND : BOOL;
		(* Generated from item 'RelationalOperator1' *)
		bRelationalOperator1 : BOOL;
		(* Generated from item 'CastToBoolean' *)
		bCastToBoolean : BOOL;
		 {attribute 'hide'}
		_reserved1 : ARRAY [1..7] OF USINT;
		(* Generated from item 'sf_MATLABFunction1' *)
		stsf_MATLABFunction1 : ST_B_MATLABFunction_vertical_levitation_control_new_T;
		(* Generated from item 'sf_MATLABFunction' *)
		stsf_MATLABFunction : ST_B_MATLABFunction_vertical_levitation_control_new_T;
	END_STRUCT
END_TYPE

// DUTs/T_ZCSigState
(* Generated from type 'ZCSigState' *)
{attribute 'TcIecLibraryType'}
TYPE T_ZCSigState : USINT;
END_TYPE

// DUTs/T_matrix4xZCSigState
(* Generated from type 'matrix4xZCSigState' *)
{attribute 'TcIecLibraryType'}
{attribute 'BaseTypeGUID' := 'CF0EC509-8CFA-173E-6D32-2A6837BC8565'}
TYPE T_matrix4xZCSigState : ARRAY [0..3] OF T_ZCSigState;
END_TYPE

// DUTs/ST_PrevZCX_vertical_levitation_control_new_T
(* Generated from type 'PrevZCX_vertical_levitation_control_new_T' *)
{attribute 'TcIecLibraryType'}
TYPE ST_PrevZCX_vertical_levitation_control_new_T : 
	STRUCT
		(* Generated from item 'Integrator1_Reset_ZCE' *)
		aIntegrator1_Reset_ZCE : T_matrix4xZCSigState;
		(* Generated from item 'Integrator_Reset_ZCE' *)
		nIntegrator_Reset_ZCE : T_ZCSigState;
		(* Generated from item 'Filter_Reset_ZCE' *)
		nFilter_Reset_ZCE : T_ZCSigState;
		(* Generated from item 'Integrator_Reset_ZCE_k' *)
		nIntegrator_Reset_ZCE_k : T_ZCSigState;
		(* Generated from item 'Filtertot_Reset_ZCE' *)
		nFiltertot_Reset_ZCE : T_ZCSigState;
		(* Generated from item 'Integrator_Reset_ZCE_m' *)
		nIntegrator_Reset_ZCE_m : T_ZCSigState;
		(* Generated from item 'Filterroll_Reset_ZCE' *)
		nFilterroll_Reset_ZCE : T_ZCSigState;
		(* Generated from item 'Integrator_Reset_ZCE_km' *)
		nIntegrator_Reset_ZCE_km : T_ZCSigState;
		(* Generated from item 'Filterpit_Reset_ZCE' *)
		nFilterpit_Reset_ZCE : T_ZCSigState;
		(* Generated from item 'Integrator_Reset_ZCE_b' *)
		nIntegrator_Reset_ZCE_b : T_ZCSigState;
		(* Generated from item 'Filter_Reset_ZCE_m' *)
		nFilter_Reset_ZCE_m : T_ZCSigState;
		(* Generated from item 'Integrator_Reset_ZCE_d' *)
		nIntegrator_Reset_ZCE_d : T_ZCSigState;
		(* Generated from item 'Filter_Reset_ZCE_a' *)
		nFilter_Reset_ZCE_a : T_ZCSigState;
		(* Generated from item 'Integrator2_Reset_ZCE' *)
		aIntegrator2_Reset_ZCE : T_matrix4xZCSigState;
	END_STRUCT
END_TYPE

// DUTs/ST_X_vertical_levitation_control_new_T
(* Generated from type 'X_vertical_levitation_control_new_T' *)
{attribute 'TcIecLibraryType'}
TYPE ST_X_vertical_levitation_control_new_T : 
	STRUCT
		(* Generated from item 'Integrator1_CSTATE' *)
		aIntegrator1_CSTATE : T_matrix4xdouble;
		(* Generated from item 'Integrator_CSTATE' *)
		fIntegrator_CSTATE : LREAL;
		(* Generated from item 'Filter_CSTATE' *)
		fFilter_CSTATE : LREAL;
		(* Generated from item 'Integrator_CSTATE_p' *)
		fIntegrator_CSTATE_p : LREAL;
		(* Generated from item 'Filtertot_CSTATE' *)
		fFiltertot_CSTATE : LREAL;
		(* Generated from item 'Integrator_CSTATE_k' *)
		fIntegrator_CSTATE_k : LREAL;
		(* Generated from item 'Filterroll_CSTATE' *)
		fFilterroll_CSTATE : LREAL;
		(* Generated from item 'Integrator_CSTATE_pl' *)
		fIntegrator_CSTATE_pl : LREAL;
		(* Generated from item 'Filterpit_CSTATE' *)
		fFilterpit_CSTATE : LREAL;
		(* Generated from item 'Integrator_CSTATE_c' *)
		fIntegrator_CSTATE_c : LREAL;
		(* Generated from item 'Filter_CSTATE_j' *)
		fFilter_CSTATE_j : LREAL;
		(* Generated from item 'Integrator_CSTATE_pq' *)
		fIntegrator_CSTATE_pq : LREAL;
		(* Generated from item 'Filter_CSTATE_b' *)
		fFilter_CSTATE_b : LREAL;
		(* Generated from item 'Integrator2_CSTATE' *)
		aIntegrator2_CSTATE : T_matrix4xdouble;
	END_STRUCT
END_TYPE

// DUTs/ST_ExtU_vertical_levitation_control_new_T
(* Generated from type 'ExtU_vertical_levitation_control_new_T' *)
{attribute 'TcIecLibraryType'}
TYPE ST_ExtU_vertical_levitation_control_new_T : 
	STRUCT
		(* Generated from item 'z_avg' *)
		fz_avg : LREAL;
		(* Generated from item 'roll_measured' *)
		froll_measured : LREAL;
		(* Generated from item 'pitch_measured' *)
		fpitch_measured : LREAL;
		(* Generated from item 'ems_roll' *)
		fems_roll : LREAL;
		(* Generated from item 'F_imu' *)
		aF_imu : T_matrix3xdouble;
		(* Generated from item 'gyro_imu' *)
		agyro_imu : T_matrix3xdouble;
		(* Generated from item 'motor_Fy_l' *)
		fmotor_Fy_l : LREAL;
		(* Generated from item 'motor_Fy_r' *)
		fmotor_Fy_r : LREAL;
	END_STRUCT
END_TYPE

// DUTs/ST_ExtY_vertical_levitation_control_new_T
(* Generated from type 'ExtY_vertical_levitation_control_new_T' *)
{attribute 'TcIecLibraryType'}
TYPE ST_ExtY_vertical_levitation_control_new_T : 
	STRUCT
		(* Generated from item 'I_VFL' *)
		aI_VFL : T_matrix2xdouble;
		(* Generated from item 'I_VFR' *)
		aI_VFR : T_matrix2xdouble;
		(* Generated from item 'I_VBL' *)
		aI_VBL : T_matrix2xdouble;
		(* Generated from item 'I_VBR' *)
		aI_VBR : T_matrix2xdouble;
		(* Generated from item 'F_hems' *)
		aF_hems : T_matrix4xdouble;
		(* Generated from item 'F_requested' *)
		aF_requested : T_matrix3xdouble;
		(* Generated from item 'integral_terms' *)
		aintegral_terms : T_matrix3xdouble;
		(* Generated from item 'sat_failed' *)
		fsat_failed : LREAL;
		(* Generated from item 'net_post_sat' *)
		anet_post_sat : T_matrix3xdouble;
		(* Generated from item 'Max_allowed_current' *)
		aMax_allowed_current : T_matrix4xdouble;
		(* Generated from item 'Min_allowed_current' *)
		aMin_allowed_current : T_matrix4xdouble;
	END_STRUCT
END_TYPE

// DUTs/T_matrix4xbool
(* Generated from type 'matrix4xbool' *)
{attribute 'TcIecLibraryType'}
{attribute 'BaseTypeGUID' := '18071995-0000-0000-0000-000000000030'}
TYPE T_matrix4xbool : ARRAY [0..3] OF BOOL;
END_TYPE

// DUTs/ST_XDis_vertical_levitation_control_new_T
(* Generated from type 'XDis_vertical_levitation_control_new_T' *)
{attribute 'TcIecLibraryType'}
TYPE ST_XDis_vertical_levitation_control_new_T : 
	STRUCT
		(* Generated from item 'Integrator1_CSTATE' *)
		aIntegrator1_CSTATE : T_matrix4xbool;
		(* Generated from item 'Integrator_CSTATE' *)
		bIntegrator_CSTATE : BOOL;
		(* Generated from item 'Filter_CSTATE' *)
		bFilter_CSTATE : BOOL;
		(* Generated from item 'Integrator_CSTATE_p' *)
		bIntegrator_CSTATE_p : BOOL;
		(* Generated from item 'Filtertot_CSTATE' *)
		bFiltertot_CSTATE : BOOL;
		(* Generated from item 'Integrator_CSTATE_k' *)
		bIntegrator_CSTATE_k : BOOL;
		(* Generated from item 'Filterroll_CSTATE' *)
		bFilterroll_CSTATE : BOOL;
		(* Generated from item 'Integrator_CSTATE_pl' *)
		bIntegrator_CSTATE_pl : BOOL;
		(* Generated from item 'Filterpit_CSTATE' *)
		bFilterpit_CSTATE : BOOL;
		(* Generated from item 'Integrator_CSTATE_c' *)
		bIntegrator_CSTATE_c : BOOL;
		(* Generated from item 'Filter_CSTATE_j' *)
		bFilter_CSTATE_j : BOOL;
		(* Generated from item 'Integrator_CSTATE_pq' *)
		bIntegrator_CSTATE_pq : BOOL;
		(* Generated from item 'Filter_CSTATE_b' *)
		bFilter_CSTATE_b : BOOL;
		(* Generated from item 'Integrator2_CSTATE' *)
		aIntegrator2_CSTATE : T_matrix4xbool;
	END_STRUCT
END_TYPE

// DUTs/T_matrix20xdouble
(* Generated from type 'matrix20xdouble' *)
{attribute 'TcIecLibraryType'}
TYPE T_matrix20xdouble : ARRAY [0..19] OF LREAL;
END_TYPE

// DUTs/T_matrix20x4xdouble
(* Generated from type 'matrix20x4xdouble' *)
{attribute 'TcIecLibraryType'}
TYPE T_matrix20x4xdouble : ARRAY [0..3,0..19] OF LREAL;
END_TYPE

// DUTs/PLREAL
{attribute 'TcIecLibraryType'}
TYPE PLREAL : POINTER TO LREAL;
END_TYPE

// DUTs/T_matrix4xdoublepointer
(* Generated from type 'matrix4xdouble *' *)
{attribute 'TcIecLibraryType'}
{attribute 'BaseTypeGUID' := '2CE33DB5-EBD3-49F7-1FA0-F8105FFA7B54'}
TYPE T_matrix4xdoublepointer : ARRAY [0..3] OF PLREAL;
END_TYPE

// DUTs/ST_ODE4_IntgData
(* Generated from type 'ODE4_IntgData' *)
{attribute 'TcIecLibraryType'}
{attribute 'pack_mode' := '1'}
TYPE ST_ODE4_IntgData : 
	STRUCT
		y : POINTER TO LREAL;
		(* Generated from item 'f' *)
		af : T_matrix4xdoublepointer;
	END_STRUCT
END_TYPE

// DUTs/ST_DW_vertical_levitation_control_new_T
(* Generated from type 'DW_vertical_levitation_control_new_T' *)
{attribute 'TcIecLibraryType'}
TYPE ST_DW_vertical_levitation_control_new_T : 
	STRUCT
		(* Generated from item 'UnitDelay_DSTATE' *)
		aUnitDelay_DSTATE : T_matrix4xdouble;
		(* Generated from item 'Delay_DSTATE' *)
		aDelay_DSTATE : T_matrix3xdouble;
		(* Generated from item 'UnitDelay1_DSTATE' *)
		fUnitDelay1_DSTATE : LREAL;
		(* Generated from item 'UnitDelay1_DSTATE_f' *)
		fUnitDelay1_DSTATE_f : LREAL;
		(* Generated from item 'UnitDelay1_DSTATE_i' *)
		fUnitDelay1_DSTATE_i : LREAL;
		(* Generated from item 'UnitDelay1_DSTATE_j' *)
		fUnitDelay1_DSTATE_j : LREAL;
		(* Generated from item 'UnitDelay1_DSTATE_m' *)
		fUnitDelay1_DSTATE_m : LREAL;
		(* Generated from item 'UnitDelay1_DSTATE_d' *)
		fUnitDelay1_DSTATE_d : LREAL;
		(* Generated from item 'UnitDelay1_DSTATE_mr' *)
		fUnitDelay1_DSTATE_mr : LREAL;
		(* Generated from item 'UnitDelay1_DSTATE_e' *)
		fUnitDelay1_DSTATE_e : LREAL;
		(* Generated from item 'UD_DSTATE' *)
		fUD_DSTATE : LREAL;
		(* Generated from item 'UnitDelay1_DSTATE_mp' *)
		fUnitDelay1_DSTATE_mp : LREAL;
		(* Generated from item 'UnitDelay1_DSTATE_a' *)
		fUnitDelay1_DSTATE_a : LREAL;
		(* Generated from item 'UnitDelay1_DSTATE_p' *)
		fUnitDelay1_DSTATE_p : LREAL;
		(* Generated from item 'UnitDelay1_DSTATE_g' *)
		fUnitDelay1_DSTATE_g : LREAL;
		(* Generated from item 'UnitDelay1_DSTATE_f3' *)
		fUnitDelay1_DSTATE_f3 : LREAL;
		(* Generated from item 'UnitDelay1_DSTATE_ab' *)
		fUnitDelay1_DSTATE_ab : LREAL;
		(* Generated from item 'UnitDelay1_DSTATE_ia' *)
		fUnitDelay1_DSTATE_ia : LREAL;
		(* Generated from item 'UnitDelay1_DSTATE_o' *)
		fUnitDelay1_DSTATE_o : LREAL;
		(* Generated from item 'UnitDelay1_DSTATE_ed' *)
		fUnitDelay1_DSTATE_ed : LREAL;
		(* Generated from item 'UnitDelay1_DSTATE_ei' *)
		fUnitDelay1_DSTATE_ei : LREAL;
		(* Generated from item 'UnitDelay1_DSTATE_b' *)
		fUnitDelay1_DSTATE_b : LREAL;
		(* Generated from item 'UnitDelay1_DSTATE_bj' *)
		fUnitDelay1_DSTATE_bj : LREAL;
		(* Generated from item 'UnitDelay1_DSTATE_ph' *)
		fUnitDelay1_DSTATE_ph : LREAL;
		(* Generated from item 'UnitDelay1_DSTATE_as' *)
		fUnitDelay1_DSTATE_as : LREAL;
		(* Generated from item 'UnitDelay1_DSTATE_c' *)
		fUnitDelay1_DSTATE_c : LREAL;
		(* Generated from item 'UnitDelay1_DSTATE_dj' *)
		fUnitDelay1_DSTATE_dj : LREAL;
		(* Generated from item 'UnitDelay2_DSTATE' *)
		fUnitDelay2_DSTATE : LREAL;
		(* Generated from item 'UnitDelay2_DSTATE_l' *)
		fUnitDelay2_DSTATE_l : LREAL;
		(* Generated from item 'UnitDelay2_DSTATE_l5' *)
		fUnitDelay2_DSTATE_l5 : LREAL;
		(* Generated from item 'UnitDelay2_DSTATE_i' *)
		fUnitDelay2_DSTATE_i : LREAL;
		(* Generated from item 'UnitDelay2_DSTATE_c' *)
		fUnitDelay2_DSTATE_c : LREAL;
		(* Generated from item 'UnitDelay2_DSTATE_d' *)
		fUnitDelay2_DSTATE_d : LREAL;
		(* Generated from item 'UnitDelay2_DSTATE_f' *)
		fUnitDelay2_DSTATE_f : LREAL;
		(* Generated from item 'UnitDelay2_DSTATE_iz' *)
		fUnitDelay2_DSTATE_iz : LREAL;
		(* Generated from item 'UnitDelay2_DSTATE_n' *)
		fUnitDelay2_DSTATE_n : LREAL;
		(* Generated from item 'UnitDelay2_DSTATE_p' *)
		fUnitDelay2_DSTATE_p : LREAL;
		(* Generated from item 'UnitDelay2_DSTATE_l0' *)
		fUnitDelay2_DSTATE_l0 : LREAL;
		(* Generated from item 'UnitDelay2_DSTATE_b' *)
		fUnitDelay2_DSTATE_b : LREAL;
		(* Generated from item 'UnitDelay2_DSTATE_g' *)
		fUnitDelay2_DSTATE_g : LREAL;
		(* Generated from item 'UnitDelay2_DSTATE_k' *)
		fUnitDelay2_DSTATE_k : LREAL;
		(* Generated from item 'UnitDelay2_DSTATE_fe' *)
		fUnitDelay2_DSTATE_fe : LREAL;
		(* Generated from item 'UnitDelay2_DSTATE_fz' *)
		fUnitDelay2_DSTATE_fz : LREAL;
		(* Generated from item 'UnitDelay2_DSTATE_gi' *)
		fUnitDelay2_DSTATE_gi : LREAL;
		(* Generated from item 'UnitDelay2_DSTATE_ih' *)
		fUnitDelay2_DSTATE_ih : LREAL;
		(* Generated from item 'UnitDelay2_DSTATE_l5x' *)
		fUnitDelay2_DSTATE_l5x : LREAL;
		(* Generated from item 'UnitDelay2_DSTATE_a' *)
		fUnitDelay2_DSTATE_a : LREAL;
		(* Generated from item 'UnitDelay2_DSTATE_aa' *)
		fUnitDelay2_DSTATE_aa : LREAL;
		(* Generated from item 'Delay1_DSTATE' *)
		fDelay1_DSTATE : REAL;
		(* Generated from item 'Memory_PreviousInput' *)
		bMemory_PreviousInput : BOOL;
		(* Generated from item 'Memory_PreviousInput_l' *)
		bMemory_PreviousInput_l : BOOL;
		(* Generated from item 'Memory_PreviousInput_a' *)
		bMemory_PreviousInput_a : BOOL;
		 {attribute 'hide'}
		_reserved1 : USINT;
	END_STRUCT
END_TYPE

// DUTs/ST_x08a7a7bbd0e5d629f7d70ceec84eacfe
(* Generated from type 'x08a7a7bbd0e5d629f7d70ceec84eacfe' *)
{attribute 'TcIecLibraryType'}
TYPE ST_x08a7a7bbd0e5d629f7d70ceec84eacfe : 
	STRUCT
		(* Generated from item 'numContStates' *)
		nnumContStates : DINT;
		(* Generated from item 'numPeriodicContStates' *)
		nnumPeriodicContStates : DINT;
		(* Generated from item 'numSampTimes' *)
		nnumSampTimes : DINT;
	END_STRUCT
END_TYPE

// DUTs/ST_xf09845edab6c83520d8d57def6d6fe1c
(* Generated from type 'xf09845edab6c83520d8d57def6d6fe1c' *)
{attribute 'TcIecLibraryType'}
TYPE ST_xf09845edab6c83520d8d57def6d6fe1c : 
	STRUCT
		(* Generated from item 'clockTick0' *)
		nclockTick0 : UDINT;
		(* Generated from item 'clockTickH0' *)
		nclockTickH0 : UDINT;
		(* Generated from item 'stepSize0' *)
		fstepSize0 : LREAL;
		(* Generated from item 'clockTick1' *)
		nclockTick1 : UDINT;
		(* Generated from item 'clockTickH1' *)
		nclockTickH1 : UDINT;
		(* Generated from item 'tStart' *)
		ftStart : LREAL;
		(* Generated from item 'simTimeStep' *)
		esimTimeStep : E_SimTimeStep;
		(* Generated from item 'stopRequestedFlag' *)
		bstopRequestedFlag : BOOL;
		 {attribute 'hide'}
		_reserved1 : ARRAY [1..3] OF USINT;
		t : POINTER TO LREAL;
		(* Generated from item 'tArray' *)
		atArray : T_matrix2xdouble;
	END_STRUCT
END_TYPE

// DUTs/ST_RT_MODEL_vertical_levitation_control_new_T
(* Generated from type 'RT_MODEL_vertical_levitation_control_new_T' *)
{attribute 'TcIecLibraryType'}
{attribute 'pack_mode' := '1'}
TYPE ST_RT_MODEL_vertical_levitation_control_new_T : 
	STRUCT
		errorStatus : POINTER TO SINT;
		solverInfo : POINTER TO ST_ssSolverInfo;
		blockIO : POINTER TO ST_B_vertical_levitation_control_new_T;
		prevZCSigState : POINTER TO ST_PrevZCX_vertical_levitation_control_new_T;
		contStates : POINTER TO ST_X_vertical_levitation_control_new_T;
		periodicContStateIndices : POINTER TO DINT;
		periodicContStateRanges : POINTER TO LREAL;
		derivs : POINTER TO LREAL;
		inputs : POINTER TO ST_ExtU_vertical_levitation_control_new_T;
		outputs : POINTER TO ST_ExtY_vertical_levitation_control_new_T;
		contStateDisabled : POINTER TO ST_XDis_vertical_levitation_control_new_T;
		(* Generated from item 'zCCacheNeedsReset' *)
		bzCCacheNeedsReset : BOOL;
		(* Generated from item 'derivCacheNeedsReset' *)
		bderivCacheNeedsReset : BOOL;
		(* Generated from item 'CTOutputIncnstWithState' *)
		bCTOutputIncnstWithState : BOOL;
		 {attribute 'hide'}
		_reserved1 : UINT_8_40;
		(* Generated from item 'odeY' *)
		aodeY : T_matrix20xdouble;
		(* Generated from item 'odeF' *)
		aodeF : T_matrix20x4xdouble;
		(* Generated from item 'intgData' *)
		stintgData : ST_ODE4_IntgData;
		dwork : POINTER TO ST_DW_vertical_levitation_control_new_T;
		(* Generated from item 'Sizes' *)
		stSizes : ST_x08a7a7bbd0e5d629f7d70ceec84eacfe;
		 {attribute 'hide'}
		_reserved2 : UDINT;
		(* Generated from item 'Timing' *)
		stTiming : ST_xf09845edab6c83520d8d57def6d6fe1c;
	END_STRUCT
END_TYPE

// DUTs/T_matrix53xdouble
(* Generated from type 'matrix53xdouble' *)
{attribute 'TcIecLibraryType'}
TYPE T_matrix53xdouble : ARRAY [0..52] OF LREAL;
END_TYPE

// DUTs/T_matrix1007xdouble
(* Generated from type 'matrix1007xdouble' *)
{attribute 'TcIecLibraryType'}
TYPE T_matrix1007xdouble : ARRAY [0..1006] OF LREAL;
END_TYPE

// DUTs/T_matrix19xdouble
(* Generated from type 'matrix19xdouble' *)
{attribute 'TcIecLibraryType'}
TYPE T_matrix19xdouble : ARRAY [0..18] OF LREAL;
END_TYPE

// DUTs/T_matrix380xdouble
(* Generated from type 'matrix380xdouble' *)
{attribute 'TcIecLibraryType'}
TYPE T_matrix380xdouble : ARRAY [0..379] OF LREAL;
END_TYPE

// DUTs/T_matrix3xlogical
(* Generated from type 'matrix3xlogical' *)
{attribute 'TcIecLibraryType'}
{attribute 'BaseTypeGUID' := '18071995-0000-0000-0000-000000000030'}
TYPE T_matrix3xlogical : ARRAY [0..2] OF BOOL;
END_TYPE

// DUTs/ST_P_vertical_levitation_control_new_T
(* Generated from type 'P_vertical_levitation_control_new_T' *)
{attribute 'TcIecLibraryType'}
TYPE ST_P_vertical_levitation_control_new_T : 
	STRUCT
		(* Generated from item 'Airgaps_HEMS_DH10' *)
		aAirgaps_HEMS_DH10 : T_matrix53xdouble;
		(* Generated from item 'Current_to_force_coefficients_HEMS_DH10' *)
		aCurrent_to_force_coefficients_HEMS_DH10 : T_matrix1007xdouble;
		(* Generated from item 'Currents_HEMS_DH10' *)
		aCurrents_HEMS_DH10 : T_matrix19xdouble;
		(* Generated from item 'Force_to_current_coefficients_HEMS_DH10' *)
		aForce_to_current_coefficients_HEMS_DH10 : T_matrix380xdouble;
		(* Generated from item 'K_D_pit' *)
		fK_D_pit : LREAL;
		(* Generated from item 'K_D_roll' *)
		fK_D_roll : LREAL;
		(* Generated from item 'K_D_tot' *)
		fK_D_tot : LREAL;
		(* Generated from item 'K_F_init_pit' *)
		fK_F_init_pit : LREAL;
		(* Generated from item 'K_F_init_roll' *)
		fK_F_init_roll : LREAL;
		(* Generated from item 'K_F_init_tot' *)
		fK_F_init_tot : LREAL;
		(* Generated from item 'K_F_pit' *)
		fK_F_pit : LREAL;
		(* Generated from item 'K_F_roll' *)
		fK_F_roll : LREAL;
		(* Generated from item 'K_F_tot' *)
		fK_F_tot : LREAL;
		(* Generated from item 'K_I_init_pit' *)
		fK_I_init_pit : LREAL;
		(* Generated from item 'K_I_init_roll' *)
		fK_I_init_roll : LREAL;
		(* Generated from item 'K_I_init_tot' *)
		fK_I_init_tot : LREAL;
		(* Generated from item 'K_I_pit' *)
		fK_I_pit : LREAL;
		(* Generated from item 'K_I_roll' *)
		fK_I_roll : LREAL;
		(* Generated from item 'K_I_tot' *)
		fK_I_tot : LREAL;
		(* Generated from item 'K_P_pit' *)
		fK_P_pit : LREAL;
		(* Generated from item 'K_P_roll' *)
		fK_P_roll : LREAL;
		(* Generated from item 'K_P_tot' *)
		fK_P_tot : LREAL;
		(* Generated from item 'd_HEMS_to_HEMS' *)
		fd_HEMS_to_HEMS : LREAL;
		(* Generated from item 'f_extra_pitch_filter_1' *)
		ff_extra_pitch_filter_1 : LREAL;
		(* Generated from item 'f_extra_pitch_filter_2' *)
		ff_extra_pitch_filter_2 : LREAL;
		(* Generated from item 'f_extra_pitch_filter_3' *)
		ff_extra_pitch_filter_3 : LREAL;
		(* Generated from item 'f_extra_roll_filter_1' *)
		ff_extra_roll_filter_1 : LREAL;
		(* Generated from item 'f_extra_roll_filter_2' *)
		ff_extra_roll_filter_2 : LREAL;
		(* Generated from item 'f_extra_roll_filter_3' *)
		ff_extra_roll_filter_3 : LREAL;
		(* Generated from item 'f_extra_total_filter_1' *)
		ff_extra_total_filter_1 : LREAL;
		(* Generated from item 'f_extra_total_filter_2' *)
		ff_extra_total_filter_2 : LREAL;
		(* Generated from item 'f_extra_total_filter_3' *)
		ff_extra_total_filter_3 : LREAL;
		(* Generated from item 'f_vert_notch_main_1' *)
		ff_vert_notch_main_1 : LREAL;
		(* Generated from item 'f_vert_notch_main_2' *)
		ff_vert_notch_main_2 : LREAL;
		(* Generated from item 'f_vert_notch_main_3' *)
		ff_vert_notch_main_3 : LREAL;
		(* Generated from item 'f_vert_notch_main_4' *)
		ff_vert_notch_main_4 : LREAL;
		(* Generated from item 'g' *)
		fg : LREAL;
		(* Generated from item 'hems_under_gap' *)
		fhems_under_gap : LREAL;
		(* Generated from item 'm' *)
		fm : LREAL;
		(* Generated from item 'motor_roll_gain' *)
		fmotor_roll_gain : LREAL;
		(* Generated from item 'notch_damp' *)
		fnotch_damp : LREAL;
		(* Generated from item 'notch_gmin' *)
		fnotch_gmin : LREAL;
		(* Generated from item 'pitch_target' *)
		fpitch_target : LREAL;
		(* Generated from item 'r_motor_left_com' *)
		ar_motor_left_com : T_matrix3xdouble;
		(* Generated from item 'r_motor_right_com' *)
		ar_motor_right_com : T_matrix3xdouble;
		(* Generated from item 'r_pitch_hems' *)
		ar_pitch_hems : T_matrix4xdouble;
		(* Generated from item 'r_roll_hems' *)
		ar_roll_hems : T_matrix4xdouble;
		(* Generated from item 'roll_target' *)
		froll_target : LREAL;
		(* Generated from item 'thermal_gap_gain_hems' *)
		fthermal_gap_gain_hems : LREAL;
		(* Generated from item 'wheel_compression_liftoff' *)
		fwheel_compression_liftoff : LREAL;
		(* Generated from item 'z_initial_lift_off' *)
		fz_initial_lift_off : LREAL;
		(* Generated from item 'z_manual_target' *)
		fz_manual_target : LREAL;
		(* Generated from item 'z_mismatch_D' *)
		fz_mismatch_D : LREAL;
		(* Generated from item 'z_mismatch_F' *)
		fz_mismatch_F : LREAL;
		(* Generated from item 'z_mismatch_I' *)
		fz_mismatch_I : LREAL;
		(* Generated from item 'z_mismatch_P' *)
		fz_mismatch_P : LREAL;
		(* Generated from item 'enable_extra_pitch_notch_1' *)
		benable_extra_pitch_notch_1 : BOOL;
		(* Generated from item 'enable_extra_pitch_notch_2' *)
		benable_extra_pitch_notch_2 : BOOL;
		(* Generated from item 'enable_extra_pitch_notch_3' *)
		benable_extra_pitch_notch_3 : BOOL;
		(* Generated from item 'enable_extra_roll_notch_1' *)
		benable_extra_roll_notch_1 : BOOL;
		(* Generated from item 'enable_extra_roll_notch_2' *)
		benable_extra_roll_notch_2 : BOOL;
		(* Generated from item 'enable_extra_roll_notch_3' *)
		benable_extra_roll_notch_3 : BOOL;
		(* Generated from item 'enable_extra_total_notch_1' *)
		benable_extra_total_notch_1 : BOOL;
		(* Generated from item 'enable_extra_total_notch_2' *)
		benable_extra_total_notch_2 : BOOL;
		(* Generated from item 'enable_extra_total_notch_3' *)
		benable_extra_total_notch_3 : BOOL;
		(* Generated from item 'enable_vert_main_notch_1' *)
		benable_vert_main_notch_1 : BOOL;
		(* Generated from item 'enable_vert_main_notch_2' *)
		benable_vert_main_notch_2 : BOOL;
		(* Generated from item 'enable_vert_main_notch_3' *)
		benable_vert_main_notch_3 : BOOL;
		(* Generated from item 'enable_vert_main_notch_4' *)
		benable_vert_main_notch_4 : BOOL;
		(* Generated from item 'feed_forward_ems_ON' *)
		bfeed_forward_ems_ON : BOOL;
		(* Generated from item 'feed_fwd_motor_roll_ON' *)
		bfeed_fwd_motor_roll_ON : BOOL;
		(* Generated from item 'levi_operational' *)
		blevi_operational : BOOL;
		(* Generated from item 'mismatch_enabled' *)
		bmismatch_enabled : BOOL;
		(* Generated from item 'mismatch_specific_enabler' *)
		amismatch_specific_enabler : T_matrix3xlogical;
		(* Generated from item 'pitch_ON' *)
		bpitch_ON : BOOL;
		(* Generated from item 'roll_ON' *)
		broll_ON : BOOL;
		(* Generated from item 'roll_filter_enabled' *)
		broll_filter_enabled : BOOL;
		(* Generated from item 'total_ON' *)
		btotal_ON : BOOL;
		(* Generated from item 'DiscreteDerivative_ICPrevScaledInput' *)
		fDiscreteDerivative_ICPrevScaledInput : LREAL;
		(* Generated from item 'PIDController_InitialConditionForFilter' *)
		fPIDController_InitialConditionForFilter : LREAL;
		(* Generated from item 'PIDController_InitialConditionForFilter_a' *)
		fPIDController_InitialConditionForFilter_a : LREAL;
		(* Generated from item 'PIDController_InitialConditionForFilter_j' *)
		fPIDController_InitialConditionForFilter_j : LREAL;
		(* Generated from item 'PIDController_InitialConditionForIntegrator' *)
		fPIDController_InitialConditionForIntegrator : LREAL;
		(* Generated from item 'PIDController_InitialConditionForIntegrator_m' *)
		fPIDController_InitialConditionForIntegrator_m : LREAL;
		(* Generated from item 'PIDController_InitialConditionForIntegrator_p' *)
		fPIDController_InitialConditionForIntegrator_p : LREAL;
		(* Generated from item 'PIDController_LowerSaturationLimit' *)
		fPIDController_LowerSaturationLimit : LREAL;
		(* Generated from item 'PIDController_LowerSaturationLimit_n' *)
		fPIDController_LowerSaturationLimit_n : LREAL;
		(* Generated from item 'PIDController_LowerSaturationLimit_e' *)
		fPIDController_LowerSaturationLimit_e : LREAL;
		(* Generated from item 'PIDController_UpperSaturationLimit' *)
		fPIDController_UpperSaturationLimit : LREAL;
		(* Generated from item 'PIDController_UpperSaturationLimit_n' *)
		fPIDController_UpperSaturationLimit_n : LREAL;
		(* Generated from item 'PIDController_UpperSaturationLimit_g' *)
		fPIDController_UpperSaturationLimit_g : LREAL;
		(* Generated from item 'Constant1_Value' *)
		fConstant1_Value : LREAL;
		(* Generated from item 'Constant1_Value_b' *)
		fConstant1_Value_b : LREAL;
		(* Generated from item 'Constant1_Value_e' *)
		fConstant1_Value_e : LREAL;
		(* Generated from item 'Constant4_Value' *)
		fConstant4_Value : LREAL;
		(* Generated from item 'Constant4_Value_e' *)
		fConstant4_Value_e : LREAL;
		(* Generated from item 'UnitDelay_InitialCondition' *)
		fUnitDelay_InitialCondition : LREAL;
		(* Generated from item 'Integrator1_IC' *)
		fIntegrator1_IC : LREAL;
		(* Generated from item 'Constant5_Value' *)
		fConstant5_Value : LREAL;
		(* Generated from item 'Switch1_Threshold' *)
		fSwitch1_Threshold : LREAL;
		(* Generated from item 'Constant7_Value' *)
		fConstant7_Value : LREAL;
		(* Generated from item 'Switch1_Threshold_i' *)
		fSwitch1_Threshold_i : LREAL;
		(* Generated from item 'sat_enabled_Value' *)
		fsat_enabled_Value : LREAL;
		(* Generated from item 'Constant8_Value' *)
		fConstant8_Value : LREAL;
		(* Generated from item 'Constant9_Value' *)
		fConstant9_Value : LREAL;
		(* Generated from item 'Switch2_Threshold' *)
		fSwitch2_Threshold : LREAL;
		(* Generated from item 'Delay_InitialCondition' *)
		fDelay_InitialCondition : LREAL;
		(* Generated from item 'UnitDelay1_InitialCondition' *)
		fUnitDelay1_InitialCondition : LREAL;
		(* Generated from item 'Constant_Value' *)
		fConstant_Value : LREAL;
		(* Generated from item 'stop_div_by_zero_Threshold' *)
		fstop_div_by_zero_Threshold : LREAL;
		(* Generated from item 'tau_Gain' *)
		ftau_Gain : LREAL;
		(* Generated from item 'Bias_Bias' *)
		fBias_Bias : LREAL;
		(* Generated from item 'two_Gain' *)
		ftwo_Gain : LREAL;
		(* Generated from item 'one_Gain' *)
		fone_Gain : LREAL;
		(* Generated from item 'UnitDelay1_InitialCondition_n' *)
		fUnitDelay1_InitialCondition_n : LREAL;
		(* Generated from item 'tau_Gain_m' *)
		ftau_Gain_m : LREAL;
		(* Generated from item 'Bias_Bias_c' *)
		fBias_Bias_c : LREAL;
		(* Generated from item 'two_Gain_f' *)
		ftwo_Gain_f : LREAL;
		(* Generated from item 'one_Gain_k' *)
		fone_Gain_k : LREAL;
		(* Generated from item 'UnitDelay1_InitialCondition_a' *)
		fUnitDelay1_InitialCondition_a : LREAL;
		(* Generated from item 'tau_Gain_d' *)
		ftau_Gain_d : LREAL;
		(* Generated from item 'Bias_Bias_d' *)
		fBias_Bias_d : LREAL;
		(* Generated from item 'two_Gain_a' *)
		ftwo_Gain_a : LREAL;
		(* Generated from item 'one_Gain_j' *)
		fone_Gain_j : LREAL;
		(* Generated from item 'UnitDelay1_InitialCondition_d' *)
		fUnitDelay1_InitialCondition_d : LREAL;
		(* Generated from item 'tau_Gain_b' *)
		ftau_Gain_b : LREAL;
		(* Generated from item 'Bias_Bias_i' *)
		fBias_Bias_i : LREAL;
		(* Generated from item 'two_Gain_ar' *)
		ftwo_Gain_ar : LREAL;
		(* Generated from item 'one_Gain_p' *)
		fone_Gain_p : LREAL;
		(* Generated from item 'UnitDelay1_InitialCondition_m' *)
		fUnitDelay1_InitialCondition_m : LREAL;
		(* Generated from item 'tau_Gain_l' *)
		ftau_Gain_l : LREAL;
		(* Generated from item 'Bias_Bias_k' *)
		fBias_Bias_k : LREAL;
		(* Generated from item 'two_Gain_g' *)
		ftwo_Gain_g : LREAL;
		(* Generated from item 'one_Gain_pt' *)
		fone_Gain_pt : LREAL;
		(* Generated from item 'UnitDelay1_InitialCondition_c' *)
		fUnitDelay1_InitialCondition_c : LREAL;
		(* Generated from item 'tau_Gain_c' *)
		ftau_Gain_c : LREAL;
		(* Generated from item 'Bias_Bias_ib' *)
		fBias_Bias_ib : LREAL;
		(* Generated from item 'two_Gain_i' *)
		ftwo_Gain_i : LREAL;
		(* Generated from item 'one_Gain_f' *)
		fone_Gain_f : LREAL;
		(* Generated from item 'UnitDelay1_InitialCondition_k' *)
		fUnitDelay1_InitialCondition_k : LREAL;
		(* Generated from item 'tau_Gain_k' *)
		ftau_Gain_k : LREAL;
		(* Generated from item 'Bias_Bias_l' *)
		fBias_Bias_l : LREAL;
		(* Generated from item 'two_Gain_j' *)
		ftwo_Gain_j : LREAL;
		(* Generated from item 'one_Gain_l' *)
		fone_Gain_l : LREAL;
		(* Generated from item 'UnitDelay1_InitialCondition_a4' *)
		fUnitDelay1_InitialCondition_a4 : LREAL;
		(* Generated from item 'TSamp_WtEt' *)
		fTSamp_WtEt : LREAL;
		(* Generated from item 'Gain_Gain' *)
		fGain_Gain : LREAL;
		(* Generated from item 'tau_Gain_d1' *)
		ftau_Gain_d1 : LREAL;
		(* Generated from item 'Bias_Bias_e' *)
		fBias_Bias_e : LREAL;
		(* Generated from item 'two_Gain_e' *)
		ftwo_Gain_e : LREAL;
		(* Generated from item 'one_Gain_m' *)
		fone_Gain_m : LREAL;
		(* Generated from item 'UnitDelay1_InitialCondition_b' *)
		fUnitDelay1_InitialCondition_b : LREAL;
		(* Generated from item 'tau_Gain_o' *)
		ftau_Gain_o : LREAL;
		(* Generated from item 'Bias_Bias_m' *)
		fBias_Bias_m : LREAL;
		(* Generated from item 'two_Gain_ir' *)
		ftwo_Gain_ir : LREAL;
		(* Generated from item 'one_Gain_pa' *)
		fone_Gain_pa : LREAL;
		(* Generated from item 'UnitDelay1_InitialCondition_g' *)
		fUnitDelay1_InitialCondition_g : LREAL;
		(* Generated from item 'tau_Gain_e' *)
		ftau_Gain_e : LREAL;
		(* Generated from item 'Bias_Bias_kd' *)
		fBias_Bias_kd : LREAL;
		(* Generated from item 'two_Gain_i5' *)
		ftwo_Gain_i5 : LREAL;
		(* Generated from item 'one_Gain_kr' *)
		fone_Gain_kr : LREAL;
		(* Generated from item 'UnitDelay1_InitialCondition_h' *)
		fUnitDelay1_InitialCondition_h : LREAL;
		(* Generated from item 'tau_Gain_l4' *)
		ftau_Gain_l4 : LREAL;
		(* Generated from item 'Bias_Bias_a' *)
		fBias_Bias_a : LREAL;
		(* Generated from item 'two_Gain_c' *)
		ftwo_Gain_c : LREAL;
		(* Generated from item 'one_Gain_ptp' *)
		fone_Gain_ptp : LREAL;
		(* Generated from item 'UnitDelay1_InitialCondition_f' *)
		fUnitDelay1_InitialCondition_f : LREAL;
		(* Generated from item 'tau_Gain_me' *)
		ftau_Gain_me : LREAL;
		(* Generated from item 'Bias_Bias_b' *)
		fBias_Bias_b : LREAL;
		(* Generated from item 'two_Gain_o' *)
		ftwo_Gain_o : LREAL;
		(* Generated from item 'one_Gain_n' *)
		fone_Gain_n : LREAL;
		(* Generated from item 'UnitDelay1_InitialCondition_g3' *)
		fUnitDelay1_InitialCondition_g3 : LREAL;
		(* Generated from item 'tau_Gain_l4v' *)
		ftau_Gain_l4v : LREAL;
		(* Generated from item 'Bias_Bias_mg' *)
		fBias_Bias_mg : LREAL;
		(* Generated from item 'two_Gain_n' *)
		ftwo_Gain_n : LREAL;
		(* Generated from item 'one_Gain_f1' *)
		fone_Gain_f1 : LREAL;
		(* Generated from item 'UnitDelay1_InitialCondition_f5' *)
		fUnitDelay1_InitialCondition_f5 : LREAL;
		(* Generated from item 'tau_Gain_by' *)
		ftau_Gain_by : LREAL;
		(* Generated from item 'Bias_Bias_n' *)
		fBias_Bias_n : LREAL;
		(* Generated from item 'two_Gain_jg' *)
		ftwo_Gain_jg : LREAL;
		(* Generated from item 'one_Gain_o' *)
		fone_Gain_o : LREAL;
		(* Generated from item 'UnitDelay1_InitialCondition_cz' *)
		fUnitDelay1_InitialCondition_cz : LREAL;
		(* Generated from item 'Gain1_Gain' *)
		fGain1_Gain : LREAL;
		(* Generated from item 'tau_Gain_f' *)
		ftau_Gain_f : LREAL;
		(* Generated from item 'Bias_Bias_f' *)
		fBias_Bias_f : LREAL;
		(* Generated from item 'two_Gain_al' *)
		ftwo_Gain_al : LREAL;
		(* Generated from item 'one_Gain_g' *)
		fone_Gain_g : LREAL;
		(* Generated from item 'UnitDelay1_InitialCondition_l' *)
		fUnitDelay1_InitialCondition_l : LREAL;
		(* Generated from item 'tau_Gain_a' *)
		ftau_Gain_a : LREAL;
		(* Generated from item 'Bias_Bias_cu' *)
		fBias_Bias_cu : LREAL;
		(* Generated from item 'two_Gain_ji' *)
		ftwo_Gain_ji : LREAL;
		(* Generated from item 'one_Gain_fw' *)
		fone_Gain_fw : LREAL;
		(* Generated from item 'UnitDelay1_InitialCondition_h5' *)
		fUnitDelay1_InitialCondition_h5 : LREAL;
		(* Generated from item 'tau_Gain_g' *)
		ftau_Gain_g : LREAL;
		(* Generated from item 'Bias_Bias_aw' *)
		fBias_Bias_aw : LREAL;
		(* Generated from item 'two_Gain_k' *)
		ftwo_Gain_k : LREAL;
		(* Generated from item 'one_Gain_c' *)
		fone_Gain_c : LREAL;
		(* Generated from item 'UnitDelay1_InitialCondition_p' *)
		fUnitDelay1_InitialCondition_p : LREAL;
		(* Generated from item 'tau_Gain_ld' *)
		ftau_Gain_ld : LREAL;
		(* Generated from item 'Bias_Bias_mo' *)
		fBias_Bias_mo : LREAL;
		(* Generated from item 'two_Gain_of' *)
		ftwo_Gain_of : LREAL;
		(* Generated from item 'one_Gain_b' *)
		fone_Gain_b : LREAL;
		(* Generated from item 'UnitDelay1_InitialCondition_k3' *)
		fUnitDelay1_InitialCondition_k3 : LREAL;
		(* Generated from item 'tau_Gain_j' *)
		ftau_Gain_j : LREAL;
		(* Generated from item 'Bias_Bias_l1' *)
		fBias_Bias_l1 : LREAL;
		(* Generated from item 'two_Gain_o4' *)
		ftwo_Gain_o4 : LREAL;
		(* Generated from item 'one_Gain_oe' *)
		fone_Gain_oe : LREAL;
		(* Generated from item 'UnitDelay1_InitialCondition_o' *)
		fUnitDelay1_InitialCondition_o : LREAL;
		(* Generated from item 'tau_Gain_gg' *)
		ftau_Gain_gg : LREAL;
		(* Generated from item 'Bias_Bias_cz' *)
		fBias_Bias_cz : LREAL;
		(* Generated from item 'two_Gain_kw' *)
		ftwo_Gain_kw : LREAL;
		(* Generated from item 'one_Gain_d' *)
		fone_Gain_d : LREAL;
		(* Generated from item 'UnitDelay1_InitialCondition_pu' *)
		fUnitDelay1_InitialCondition_pu : LREAL;
		(* Generated from item 'tau_Gain_ct' *)
		ftau_Gain_ct : LREAL;
		(* Generated from item 'Bias_Bias_g' *)
		fBias_Bias_g : LREAL;
		(* Generated from item 'two_Gain_m' *)
		ftwo_Gain_m : LREAL;
		(* Generated from item 'one_Gain_ff' *)
		fone_Gain_ff : LREAL;
		(* Generated from item 'UnitDelay1_InitialCondition_bg' *)
		fUnitDelay1_InitialCondition_bg : LREAL;
		(* Generated from item 'dist_enabled_Value' *)
		fdist_enabled_Value : LREAL;
		(* Generated from item 'UnitDelay1_InitialCondition_ni' *)
		fUnitDelay1_InitialCondition_ni : LREAL;
		(* Generated from item 'Constant_Value_e' *)
		fConstant_Value_e : LREAL;
		(* Generated from item 'stop_div_by_zero_Threshold_g' *)
		fstop_div_by_zero_Threshold_g : LREAL;
		(* Generated from item 'UnitDelay1_InitialCondition_nc' *)
		fUnitDelay1_InitialCondition_nc : LREAL;
		(* Generated from item 'Constant_Value_a' *)
		fConstant_Value_a : LREAL;
		(* Generated from item 'stop_div_by_zero_Threshold_p' *)
		fstop_div_by_zero_Threshold_p : LREAL;
		(* Generated from item 'ZeroGain_Gain' *)
		fZeroGain_Gain : LREAL;
		(* Generated from item 'ZeroGain_Gain_m' *)
		fZeroGain_Gain_m : LREAL;
		(* Generated from item 'ZeroGain_Gain_a' *)
		fZeroGain_Gain_a : LREAL;
		(* Generated from item 'Bias1_Bias' *)
		fBias1_Bias : LREAL;
		(* Generated from item 'Gain_Gain_b' *)
		fGain_Gain_b : LREAL;
		(* Generated from item 'UnitDelay2_InitialCondition' *)
		fUnitDelay2_InitialCondition : LREAL;
		(* Generated from item 'Bias1_Bias_c' *)
		fBias1_Bias_c : LREAL;
		(* Generated from item 'Gain_Gain_k' *)
		fGain_Gain_k : LREAL;
		(* Generated from item 'UnitDelay2_InitialCondition_d' *)
		fUnitDelay2_InitialCondition_d : LREAL;
		(* Generated from item 'Bias1_Bias_p' *)
		fBias1_Bias_p : LREAL;
		(* Generated from item 'Gain_Gain_f' *)
		fGain_Gain_f : LREAL;
		(* Generated from item 'UnitDelay2_InitialCondition_b' *)
		fUnitDelay2_InitialCondition_b : LREAL;
		(* Generated from item 'Bias1_Bias_i' *)
		fBias1_Bias_i : LREAL;
		(* Generated from item 'Gain_Gain_fp' *)
		fGain_Gain_fp : LREAL;
		(* Generated from item 'UnitDelay2_InitialCondition_h' *)
		fUnitDelay2_InitialCondition_h : LREAL;
		(* Generated from item 'Bias1_Bias_p1' *)
		fBias1_Bias_p1 : LREAL;
		(* Generated from item 'Gain_Gain_o' *)
		fGain_Gain_o : LREAL;
		(* Generated from item 'UnitDelay2_InitialCondition_m' *)
		fUnitDelay2_InitialCondition_m : LREAL;
		(* Generated from item 'Bias1_Bias_a' *)
		fBias1_Bias_a : LREAL;
		(* Generated from item 'Gain_Gain_c' *)
		fGain_Gain_c : LREAL;
		(* Generated from item 'UnitDelay2_InitialCondition_c' *)
		fUnitDelay2_InitialCondition_c : LREAL;
		(* Generated from item 'Bias1_Bias_m' *)
		fBias1_Bias_m : LREAL;
		(* Generated from item 'Gain_Gain_p' *)
		fGain_Gain_p : LREAL;
		(* Generated from item 'UnitDelay2_InitialCondition_a' *)
		fUnitDelay2_InitialCondition_a : LREAL;
		(* Generated from item 'Bias1_Bias_f' *)
		fBias1_Bias_f : LREAL;
		(* Generated from item 'Gain_Gain_e' *)
		fGain_Gain_e : LREAL;
		(* Generated from item 'UnitDelay2_InitialCondition_c3' *)
		fUnitDelay2_InitialCondition_c3 : LREAL;
		(* Generated from item 'Bias1_Bias_mq' *)
		fBias1_Bias_mq : LREAL;
		(* Generated from item 'Gain_Gain_fs' *)
		fGain_Gain_fs : LREAL;
		(* Generated from item 'UnitDelay2_InitialCondition_f' *)
		fUnitDelay2_InitialCondition_f : LREAL;
		(* Generated from item 'Bias1_Bias_pl' *)
		fBias1_Bias_pl : LREAL;
		(* Generated from item 'Gain_Gain_e3' *)
		fGain_Gain_e3 : LREAL;
		(* Generated from item 'UnitDelay2_InitialCondition_i' *)
		fUnitDelay2_InitialCondition_i : LREAL;
		(* Generated from item 'Bias1_Bias_j' *)
		fBias1_Bias_j : LREAL;
		(* Generated from item 'Gain_Gain_br' *)
		fGain_Gain_br : LREAL;
		(* Generated from item 'UnitDelay2_InitialCondition_e' *)
		fUnitDelay2_InitialCondition_e : LREAL;
		(* Generated from item 'Bias1_Bias_e' *)
		fBias1_Bias_e : LREAL;
		(* Generated from item 'Gain_Gain_kc' *)
		fGain_Gain_kc : LREAL;
		(* Generated from item 'UnitDelay2_InitialCondition_hs' *)
		fUnitDelay2_InitialCondition_hs : LREAL;
		(* Generated from item 'Bias1_Bias_b' *)
		fBias1_Bias_b : LREAL;
		(* Generated from item 'Gain_Gain_n' *)
		fGain_Gain_n : LREAL;
		(* Generated from item 'UnitDelay2_InitialCondition_k' *)
		fUnitDelay2_InitialCondition_k : LREAL;
		(* Generated from item 'Bias1_Bias_e1' *)
		fBias1_Bias_e1 : LREAL;
		(* Generated from item 'Gain_Gain_c0' *)
		fGain_Gain_c0 : LREAL;
		(* Generated from item 'UnitDelay2_InitialCondition_c4' *)
		fUnitDelay2_InitialCondition_c4 : LREAL;
		(* Generated from item 'Bias1_Bias_bc' *)
		fBias1_Bias_bc : LREAL;
		(* Generated from item 'Gain_Gain_j' *)
		fGain_Gain_j : LREAL;
		(* Generated from item 'UnitDelay2_InitialCondition_p' *)
		fUnitDelay2_InitialCondition_p : LREAL;
		(* Generated from item 'Bias1_Bias_jn' *)
		fBias1_Bias_jn : LREAL;
		(* Generated from item 'Gain_Gain_l' *)
		fGain_Gain_l : LREAL;
		(* Generated from item 'UnitDelay2_InitialCondition_l' *)
		fUnitDelay2_InitialCondition_l : LREAL;
		(* Generated from item 'Bias1_Bias_g' *)
		fBias1_Bias_g : LREAL;
		(* Generated from item 'Gain_Gain_nb' *)
		fGain_Gain_nb : LREAL;
		(* Generated from item 'UnitDelay2_InitialCondition_da' *)
		fUnitDelay2_InitialCondition_da : LREAL;
		(* Generated from item 'Bias1_Bias_k' *)
		fBias1_Bias_k : LREAL;
		(* Generated from item 'Gain_Gain_np' *)
		fGain_Gain_np : LREAL;
		(* Generated from item 'UnitDelay2_InitialCondition_j' *)
		fUnitDelay2_InitialCondition_j : LREAL;
		(* Generated from item 'Bias1_Bias_ec' *)
		fBias1_Bias_ec : LREAL;
		(* Generated from item 'Gain_Gain_np5' *)
		fGain_Gain_np5 : LREAL;
		(* Generated from item 'UnitDelay2_InitialCondition_g' *)
		fUnitDelay2_InitialCondition_g : LREAL;
		(* Generated from item 'Bias1_Bias_o' *)
		fBias1_Bias_o : LREAL;
		(* Generated from item 'Gain_Gain_oh' *)
		fGain_Gain_oh : LREAL;
		(* Generated from item 'UnitDelay2_InitialCondition_o' *)
		fUnitDelay2_InitialCondition_o : LREAL;
		(* Generated from item 'Bias1_Bias_bf' *)
		fBias1_Bias_bf : LREAL;
		(* Generated from item 'Gain_Gain_ei' *)
		fGain_Gain_ei : LREAL;
		(* Generated from item 'UnitDelay2_InitialCondition_ir' *)
		fUnitDelay2_InitialCondition_ir : LREAL;
		(* Generated from item 'Constant10_Value' *)
		fConstant10_Value : LREAL;
		(* Generated from item 'Constant6_Value' *)
		fConstant6_Value : LREAL;
		(* Generated from item 'Constant7_Value_o' *)
		fConstant7_Value_o : LREAL;
		(* Generated from item 'Constant8_Value_h' *)
		fConstant8_Value_h : LREAL;
		(* Generated from item 'Constant9_Value_p' *)
		fConstant9_Value_p : LREAL;
		(* Generated from item 'Integrator2_IC' *)
		fIntegrator2_IC : LREAL;
		(* Generated from item 'IsPeak1_Threshold' *)
		fIsPeak1_Threshold : LREAL;
		(* Generated from item 'Switch2_Threshold_n' *)
		fSwitch2_Threshold_n : LREAL;
		(* Generated from item 'Constant2_Value' *)
		fConstant2_Value : LREAL;
		(* Generated from item 'Constant2_Value_e' *)
		fConstant2_Value_e : LREAL;
		(* Generated from item 'Constant2_Value_d' *)
		fConstant2_Value_d : LREAL;
		(* Generated from item 'Delay1_InitialCondition' *)
		fDelay1_InitialCondition : REAL;
		(* Generated from item 'wasfmenabledlastrun_Threshold' *)
		fwasfmenabledlastrun_Threshold : REAL;
		(* Generated from item 'hard_disable_fmm_Gain' *)
		fhard_disable_fmm_Gain : REAL;
		(* Generated from item 'usefmornot_Threshold' *)
		fusefmornot_Threshold : REAL;
		(* Generated from item 'Memory_InitialCondition' *)
		bMemory_InitialCondition : BOOL;
		(* Generated from item 'Memory_InitialCondition_m' *)
		bMemory_InitialCondition_m : BOOL;
		(* Generated from item 'Memory_InitialCondition_n' *)
		bMemory_InitialCondition_n : BOOL;
		 {attribute 'hide'}
		_reserved1 : ARRAY [1..5] OF USINT;
	END_STRUCT
END_TYPE

// DUTs/E_ModuleCaller
(* Generated from type 'TcMgSdk.ModuleCaller' *)
{attribute 'TcIecLibraryType'}
TYPE E_ModuleCaller : (
	CyclicTask:=0, 	(* Add to the specified cyclic caller tasks. *)
	Module:=1	(* Don't add to cyclic callers. The module can be called from other TwinCAT modules (e. g. a PLC). *)
) DINT;
END_TYPE

// DUTs/E_CallerVerification
(* Generated from type 'TcMgSdk.CallerVerification' *)
{attribute 'TcIecLibraryType'}
TYPE E_CallerVerification : (
	Default:=0, 	(* Verify the caller task only if the "ModuleCaller" parameter is set to "Module" but not when added to cyclic caller tasks. *)
	Always:=1, 	(* Always verify the caller context to prevent concurrent execution of model code and corresponding DataArea mappings. *)
	Never:=2	(* Skip caller verification to reduce execution times. *)
) DINT;
END_TYPE

// DUTs/E_StepSizeAdaptation
(* Generated from type 'TcMgSdk.StepSizeAdaptation' *)
{attribute 'TcIecLibraryType'}
TYPE E_StepSizeAdaptation : (
	RequireMatchingTaskCycleTime:=0, 	(* Don't accept task cycle times other than the Simulink step sizes. *)
	UseTaskCycleTime:=1, 	(* Adapt the Smulink step sizes to the task cycle times. *)
	UseModelStepSize:=2	(* Keep the Smulink step sizes, independent of the callers cycle time. *)
) DINT;
END_TYPE

// DUTs/E_ExecutionSequence1
(* Generated from type 'TcMgSdk.ExecutionSequence1' *)
{attribute 'TcIecLibraryType'}
TYPE E_ExecutionSequence1 : (
	UpdateBeforeOutputMapping:=0, 	(* Input mapping -> State and output update -> Output mapping -> ADS processing *)
	IoAtTaskBegin:=1	(* Input mapping -> Code execution -> Output update -> ADS processing *)
) DINT;
END_TYPE

// DUTs/E_FpExcptCtrlSet
(* Generated from type 'TcMgSdk.FpExcptCtrlSet' *)
{attribute 'TcIecLibraryType'}
TYPE E_FpExcptCtrlSet : (
	CallerExceptions:=1, 	(* Use the floating point exception settings provided by the caller *)
	ThrowExceptions:=3, 	(* Enable floating point exceptions on invalid operations and divisions by zero *)
	SuppressExceptions:=5	(* Disable floating point exceptions. *)
) USINT;
END_TYPE

// DUTs/ST_TcMatSim_ModuleGeneratorInfo
(* Generated from type 'TcMatSim.ModuleGeneratorInfo' *)
{attribute 'TcIecLibraryType'}
TYPE ST_TcMatSim_ModuleGeneratorInfo : 
	STRUCT
		(* Generated from item 'MatlabVersion' *)
		nMatlabVersion : ARRAY [0..3] OF UDINT;
		(* Generated from item 'TE140xVersion' *)
		nTE140xVersion : ARRAY [0..3] OF UDINT;
	END_STRUCT
END_TYPE

// DUTs/ST_TcMatSim_SimulinkModelInfo
(* Generated from type 'TcMatSim.SimulinkModelInfo' *)
{attribute 'TcIecLibraryType'}
TYPE ST_TcMatSim_SimulinkModelInfo : 
	STRUCT
		(* Generated from item 'ModelName' *)
		{attribute 'GUID' := '18071995-0000-0000-0000-00010000007F'}
		sModelName : STRING(127);
		(* Generated from item 'SimulinkVersion' *)
		nSimulinkVersion : ARRAY [0..3] OF UDINT;
		(* Generated from item 'ModelVersion' *)
		nModelVersion : ARRAY [0..3] OF UDINT;
		(* Generated from item 'ModelChecksum' *)
		nModelChecksum : ARRAY [0..3] OF UDINT;
	END_STRUCT
END_TYPE

// DUTs/E_ParameterSharingType
(* Generated from type 'ParameterSharingType' *)
{attribute 'TcIecLibraryType'}
TYPE E_ParameterSharingType : (
	Define:=0, 	(* This module instance defines the parameter values for all further instances of this module class. Exactly one instance of this module class must use this option. *)
	Inherit:=1	(* This module instance inherits the parameter values from the instance of this module class configured to "Define" the parameter values. Model parameters configured at this instsance are ignored. *)
) DINT;
END_TYPE

